LIN {X 0,Y 180.049,Z 440.205,A -85,B 0,C 180,E1 -25229.548,E2 -25229.548} C_VEL
LIN {X 0,Y 183.844,Z 448.858,A -85,B 0,C 180,E1 -25232.195,E2 -25232.195} C_VEL
LIN {X 0,Y 187.488,Z 458.143,A -85,B 0,C 180,E1 -25234.538,E2 -25234.538} C_VEL
LIN {X 0,Y 185.037,Z 489.842,A -85,B 0,C 180,E1 -25235.548,E2 -25235.548} C_VEL
LIN {X 0,Y 183.269,Z 507.581,A -85,B 0,C 180,E1 -25236.115,E2 -25236.115} C_VEL
LIN {X 0,Y 180.751,Z 522.405,A -85,B 0,C 180,E1 -25236.923,E2 -25236.923} C_VEL
LIN {X 0,Y 177.581,Z 535.216,A -85,B 0,C 180,E1 -25237.909,E2 -25237.909} C_VEL
LIN {X 0,Y 173.62,Z 547.959,A -85,B 0,C 180,E1 -25239.277,E2 -25239.277} C_VEL
LIN {X 0,Y 168.831,Z 560.376,A -85,B 0,C 180,E1 -25241.025,E2 -25241.025} C_VEL
LIN {X 0,Y 163.725,Z 571.725,A -85,B 0,C 180,E1 -25243.142,E2 -25243.142} C_VEL
LIN {X 0,Y 158.381,Z 582.164,A -85,B 0,C 180,E1 -25245.668,E2 -25245.668} C_VEL
LIN {X 0,Y 152.274,Z 592.549,A -85,B 0,C 180,E1 -25248.882,E2 -25248.882} C_VEL
LIN {X 0,Y 147.8,Z 599.416,A -85,B 0,C 180,E1 -25251.603,E2 -25251.603} C_VEL
LIN {X 0,Y 144.873,Z 602.943,A -85,B 0,C 180,E1 -25253.069,E2 -25253.069} C_VEL
LIN {X 0,Y 138.69,Z 608.311,A -85,B 0,C 180,E1 -25255.327,E2 -25255.327} C_VEL
LIN {X 0,Y 132.604,Z 613.141,A -85,B 0,C 180,E1 -25257.925,E2 -25257.925} C_VEL
LIN {X 0,Y 129.916,Z 615.782,A -85,B 0,C 180,E1 -25259.908,E2 -25259.908} C_VEL
LIN {X 0,Y 125.767,Z 621.093,A -85,B 0,C 180,E1 -25265.227,E2 -25265.227} C_VEL
LIN {X 0,Y 122.895,Z 624.585,A -85,B 0,C 180,E1 -25269.938,E2 -25269.938} C_VEL
LIN {X 0,Y 120.481,Z 627.978,A -85,B 0,C 180,E1 -25276.512,E2 -25276.512} C_VEL
LIN {X 0,Y 119.324,Z 629.978,A -85,B 0,C 180,E1 -25283.24,E2 -25283.24} C_VEL
LIN {X 0,Y 119.226,Z 630.634,A -85,B 0,C 180,E1 -25290.005,E2 -25290.005} C_VEL
LIN {X 0,Y 119.329,Z 629.948,A -85,B 0,C 180,E1 -25296.77,E2 -25296.77} C_VEL
LIN {X 0,Y 120.487,Z 627.918,A -85,B 0,C 180,E1 -25303.498,E2 -25303.498} C_VEL
LIN {X 0,Y 122.902,Z 624.501,A -85,B 0,C 180,E1 -25310.071,E2 -25310.071} C_VEL
LIN {X 0,Y 126.846,Z 619.596,A -85,B 0,C 180,E1 -25316.316,E2 -25316.316} C_VEL
LIN {X 0,Y 130.573,Z 614.948,A -85,B 0,C 180,E1 -25320.672,E2 -25320.672} C_VEL
LIN {X 0,Y 136.58,Z 608.007,A -85,B 0,C 180,E1 -25325.377,E2 -25325.377} C_VEL
LIN {X 0,Y 137.797,Z 606.89,A -85,B 0,C 180,E1 -25326.142,E2 -25326.142} C_VEL
LIN {X 0,Y 143.3,Z 607.92,A -85,B 0,C 180,E1 -25329.616,E2 -25329.616} C_VEL
LIN {X 0,Y 152.17,Z 608.59,A -85,B 0,C 180,E1 -25333.855,E2 -25333.855} C_VEL
LIN {X 0,Y 160.46,Z 608.435,A -85,B 0,C 180,E1 -25336.914,E2 -25336.914} C_VEL
LIN {X 0,Y 161.016,Z 608.309,A -85,B 0,C 180,E1 -25337.607,E2 -25337.607} C_VEL
LIN {X 0,Y 153.834,Z 607.574,A -85,B 0,C 180,E1 -25340.238,E2 -25340.238} C_VEL
LIN {X 0,Y 144.8,Z 605.575,A -85,B 0,C 180,E1 -25344.378,E2 -25344.378} C_VEL
LIN {X 0,Y 137.047,Z 602.404,A -85,B 0,C 180,E1 -25349.149,E2 -25349.149} C_VEL
LIN {X 0,Y 130.784,Z 598.022,A -85,B 0,C 180,E1 -25354.539,E2 -25354.539} C_VEL
LIN {X 0,Y 126.404,Z 592.364,A -85,B 0,C 180,E1 -25360.513,E2 -25360.513} C_VEL
LIN {X 0,Y 123.571,Z 585.19,A -85,B 0,C 180,E1 -25366.85,E2 -25366.85} C_VEL
LIN {X 0,Y 122.591,Z 577.538,A -85,B 0,C 180,E1 -25372.589,E2 -25372.589} C_VEL
LIN {X 0,Y 122.404,Z 569.444,A -85,B 0,C 180,E1 -25377.532,E2 -25377.532} C_VEL
LIN {X 0,Y 122.41,Z 566.355,A -85,B 0,C 180,E1 -25379.178,E2 -25379.178} C_VEL
LIN {X 0,Y 122.007,Z 566.876,A -85,B 0,C 180,E1 -25380,E2 -25380} C_VEL
LIN {X 0,Y 122.855,Z 565.896,A -85,B 0,C 180,E1 -25383.28,E2 -25383.28} C_VEL
LIN {X 0,Y 125.234,Z 563.196,A -85,B 0,C 180,E1 -25386.445,E2 -25386.445} C_VEL
LIN {X 0,Y 127.113,Z 561.789,A -85,B 0,C 180,E1 -25389.548,E2 -25389.548} C_VEL
LIN {X 0,Y 129.192,Z 559.973,A -85,B 0,C 180,E1 -25391.689,E2 -25391.689} C_VEL
LIN {X 0,Y 130.196,Z 558.96,A -85,B 0,C 180,E1 -25392.47,E2 -25392.47} C_VEL
LIN {X 0,Y 132.848,Z 557.281,A -85,B 0,C 180,E1 -25395.338,E2 -25395.338} C_VEL
LIN {X 0,Y 135.243,Z 555.329,A -85,B 0,C 180,E1 -25397.062,E2 -25397.062} C_VEL
LIN {X 0,Y 138.996,Z 551.77,A -85,B 0,C 180,E1 -25399.188,E2 -25399.188} C_VEL
LIN {X 0,Y 140.747,Z 550.664,A -85,B 0,C 180,E1 -25400.459,E2 -25400.459} C_VEL
LIN {X 0,Y 143.003,Z 548.959,A -85,B 0,C 180,E1 -25401.781,E2 -25401.781} C_VEL
LIN {X 0,Y 146.369,Z 545.737,A -85,B 0,C 180,E1 -25403.337,E2 -25403.337} C_VEL
LIN {X 0,Y 150.578,Z 541,A -85,B 0,C 180,E1 -25404.839,E2 -25404.839} C_VEL
LIN {X 0,Y 153.784,Z 538.288,A -85,B 0,C 180,E1 -25406.333,E2 -25406.333} C_VEL
LIN {X 0,Y 157.922,Z 533.92,A -85,B 0,C 180,E1 -25407.86,E2 -25407.86} C_VEL
LIN {X 0,Y 162.379,Z 527.957,A -85,B 0,C 180,E1 -25409.138,E2 -25409.138} C_VEL
LIN {X 0,Y 166.621,Z 520.75,A -85,B 0,C 180,E1 -25410.116,E2 -25410.116} C_VEL
LIN {X 0,Y 170.524,Z 512.516,A -85,B 0,C 180,E1 -25410.918,E2 -25410.918} C_VEL
LIN {X 0,Y 174.019,Z 506.932,A -85,B 0,C 180,E1 -25412.061,E2 -25412.061} C_VEL
LIN {X 0,Y 177.758,Z 499.232,A -85,B 0,C 180,E1 -25413.185,E2 -25413.185} C_VEL
LIN {X 0,Y 180.529,Z 491.731,A -85,B 0,C 180,E1 -25413.957,E2 -25413.957} C_VEL
LIN {X 0,Y 178.798,Z 507.903,A -85,B 0,C 180,E1 -25414.545,E2 -25414.545} C_VEL
LIN {X 0,Y 176.263,Z 521.664,A -85,B 0,C 180,E1 -25415.327,E2 -25415.327} C_VEL
LIN {X 0,Y 172.626,Z 535.679,A -85,B 0,C 180,E1 -25416.475,E2 -25416.475} C_VEL
LIN {X 0,Y 168.293,Z 548.682,A -85,B 0,C 180,E1 -25417.975,E2 -25417.975} C_VEL
LIN {X 0,Y 162.837,Z 561.826,A -85,B 0,C 180,E1 -25419.993,E2 -25419.993} C_VEL
LIN {X 0,Y 157.027,Z 573.992,A -85,B 0,C 180,E1 -25422.561,E2 -25422.561} C_VEL
LIN {X 0,Y 150.61,Z 585.153,A -85,B 0,C 180,E1 -25425.572,E2 -25425.572} C_VEL
LIN {X 0,Y 144.514,Z 594.607,A -85,B 0,C 180,E1 -25428.959,E2 -25428.959} C_VEL
LIN {X 0,Y 138.061,Z 603.617,A -85,B 0,C 180,E1 -25433.259,E2 -25433.259} C_VEL
LIN {X 0,Y 132.51,Z 610.879,A -85,B 0,C 180,E1 -25437.964,E2 -25437.964} C_VEL
LIN {X 0,Y 128.544,Z 615.963,A -85,B 0,C 180,E1 -25442.302,E2 -25442.302} C_VEL
LIN {X 0,Y 124.172,Z 621.222,A -85,B 0,C 180,E1 -25448.409,E2 -25448.409} C_VEL
LIN {X 0,Y 121.865,Z 624.157,A -85,B 0,C 180,E1 -25453.236,E2 -25453.236} C_VEL
LIN {X 0,Y 120.007,Z 626.851,A -85,B 0,C 180,E1 -25459.876,E2 -25459.876} C_VEL
LIN {X 0,Y 119.23,Z 628.198,A -85,B 0,C 180,E1 -25466.616,E2 -25466.616} C_VEL
LIN {X 0,Y 119.279,Z 628.373,A -85,B 0,C 180,E1 -25469.995,E2 -25469.995} C_VEL
LIN {X 0,Y 119.47,Z 627.741,A -85,B 0,C 180,E1 -25476.751,E2 -25476.751} C_VEL
LIN {X 0,Y 120.745,Z 625.774,A -85,B 0,C 180,E1 -25483.458,E2 -25483.458} C_VEL
LIN {X 0,Y 123.256,Z 622.422,A -85,B 0,C 180,E1 -25490,E2 -25490} C_VEL
LIN {X 0,Y 127.298,Z 617.581,A -85,B 0,C 180,E1 -25496.205,E2 -25496.205} C_VEL
LIN {X 0,Y 132.382,Z 611.11,A -85,B 0,C 180,E1 -25502.06,E2 -25502.06} C_VEL
LIN {X 0,Y 137.99,Z 603.902,A -85,B 0,C 180,E1 -25506.752,E2 -25506.752} C_VEL
LIN {X 0,Y 144.451,Z 594.978,A -85,B 0,C 180,E1 -25511.051,E2 -25511.051} C_VEL
LIN {X 0,Y 150.532,Z 585.604,A -85,B 0,C 180,E1 -25514.446,E2 -25514.446} C_VEL
LIN {X 0,Y 156.638,Z 575.089,A -85,B 0,C 180,E1 -25517.334,E2 -25517.334} C_VEL
LIN {X 0,Y 162.167,Z 563.764,A -85,B 0,C 180,E1 -25519.797,E2 -25519.797} C_VEL
LIN {X 0,Y 167.544,Z 551.06,A -85,B 0,C 180,E1 -25521.854,E2 -25521.854} C_VEL
LIN {X 0,Y 171.895,Z 538.676,A -85,B 0,C 180,E1 -25523.351,E2 -25523.351} C_VEL
LIN {X 0,Y 175.689,Z 524.933,A -85,B 0,C 180,E1 -25524.586,E2 -25524.586} C_VEL
LIN {X 0,Y 178.62,Z 510.582,A -85,B 0,C 180,E1 -25525.461,E2 -25525.461} C_VEL
LIN {X 0,Y 180.363,Z 496.588,A -85,B 0,C 180,E1 -25526.02,E2 -25526.02} C_VEL
LIN {X 0,Y 183.483,Z 458.98,A -85,B 0,C 180,E1 -25527.172,E2 -25527.172} C_VEL
LIN {X 0,Y 180.767,Z 452.209,A -85,B 0,C 180,E1 -25529.043,E2 -25529.043} C_VEL
LIN {X 0,Y 176.017,Z 443.177,A -85,B 0,C 180,E1 -25532.505,E2 -25532.505} C_VEL
LIN {X 0,Y 171.849,Z 436.037,A -85,B 0,C 180,E1 -25536.024,E2 -25536.024} C_VEL
LIN {X 0,Y 169.537,Z 432.413,A -85,B 0,C 180,E1 -25538.254,E2 -25538.254} C_VEL
LIN {X 0,Y 167.475,Z 429.194,A -85,B 0,C 180,E1 -25540.503,E2 -25540.503} C_VEL
LIN {X 0,Y 164.834,Z 425.188,A -85,B 0,C 180,E1 -25543.903,E2 -25543.903} C_VEL
LIN {X 0,Y 162.459,Z 421.538,A -85,B 0,C 180,E1 -25547.865,E2 -25547.865} C_VEL
LIN {X 0,Y 162.027,Z 420.886,A -85,B 0,C 180,E1 -25548.744,E2 -25548.744} C_VEL
LIN {X 0,Y 159.556,Z 415.986,A -85,B 0,C 180,E1 -25559.053,E2 -25559.053} C_VEL
LIN {X 0,Y 159.574,Z 415.731,A -85,B 0,C 180,E1 -25560.473,E2 -25560.473} C_VEL
LIN {X 0,Y 161.091,Z 419.996,A -85,B 0,C 180,E1 -25569.099,E2 -25569.099} C_VEL
LIN {X 0,Y 162.302,Z 421.185,A -85,B 0,C 180,E1 -25571.711,E2 -25571.711} C_VEL
LIN {X 0,Y 164.688,Z 425.102,A -85,B 0,C 180,E1 -25575.818,E2 -25575.818} C_VEL
LIN {X 0,Y 165.628,Z 426.451,A -85,B 0,C 180,E1 -25577.12,E2 -25577.12} C_VEL
LIN {X 0,Y 168.603,Z 430.922,A -85,B 0,C 180,E1 -25580.671,E2 -25580.671} C_VEL
LIN {X 0,Y 171.316,Z 435.2,A -85,B 0,C 180,E1 -25583.396,E2 -25583.396} C_VEL
LIN {X 0,Y 175.037,Z 441.482,A -85,B 0,C 180,E1 -25586.632,E2 -25586.632} C_VEL
LIN {X 0,Y 177.631,Z 446.437,A -85,B 0,C 180,E1 -25588.663,E2 -25588.663} C_VEL
LIN {X 0,Y 181.397,Z 455.639,A -85,B 0,C 180,E1 -25591.455,E2 -25591.455} C_VEL
LIN {X 0,Y 183.369,Z 460.941,A -85,B 0,C 180,E1 -25592.823,E2 -25592.823} C_VEL
LIN {X 0,Y 180.246,Z 498.172,A -85,B 0,C 180,E1 -25593.947,E2 -25593.947} C_VEL
LIN {X 0,Y 178.541,Z 512.168,A -85,B 0,C 180,E1 -25594.502,E2 -25594.502} C_VEL
LIN {X 0,Y 175.562,Z 526.623,A -85,B 0,C 180,E1 -25595.356,E2 -25595.356} C_VEL
LIN {X 0,Y 171.71,Z 540.435,A -85,B 0,C 180,E1 -25596.566,E2 -25596.566} C_VEL
LIN {X 0,Y 167.323,Z 552.871,A -85,B 0,C 180,E1 -25598.05,E2 -25598.05} C_VEL
LIN {X 0,Y 161.839,Z 565.623,A -85,B 0,C 180,E1 -25600.066,E2 -25600.066} C_VEL
LIN {X 0,Y 155.719,Z 577.908,A -85,B 0,C 180,E1 -25602.707,E2 -25602.707} C_VEL
LIN {X 0,Y 150.125,Z 587.55,A -85,B 0,C 180,E1 -25605.401,E2 -25605.401} C_VEL
LIN {X 0,Y 143.95,Z 596.966,A -85,B 0,C 180,E1 -25608.775,E2 -25608.775} C_VEL
LIN {X 0,Y 137.513,Z 605.936,A -85,B 0,C 180,E1 -25613.099,E2 -25613.099} C_VEL
LIN {X 0,Y 131.941,Z 613.186,A -85,B 0,C 180,E1 -25617.82,E2 -25617.82} C_VEL
LIN {X 0,Y 129.916,Z 615.782,A -85,B 0,C 180,E1 -25619.908,E2 -25619.908} C_VEL
LIN {X 0,Y 127.335,Z 618.257,A -85,B 0,C 180,E1 -25622.021,E2 -25622.021} C_VEL
LIN {X 0,Y 121.78,Z 621.8,A -85,B 0,C 180,E1 -25625.445,E2 -25625.445} C_VEL
LIN {X 0,Y 117.51,Z 624.222,A -85,B 0,C 180,E1 -25628.449,E2 -25628.449} C_VEL
LIN {X 0,Y 115.226,Z 625.795,A -85,B 0,C 180,E1 -25631.02,E2 -25631.02} C_VEL
LIN {X 0,Y 114.762,Z 626.273,A -85,B 0,C 180,E1 -25631.94,E2 -25631.94} C_VEL
LIN {X 0,Y 112.741,Z 629.081,A -85,B 0,C 180,E1 -25639.227,E2 -25639.227} C_VEL
LIN {X 0,Y 112.057,Z 630.405,A -85,B 0,C 180,E1 -25646.41,E2 -25646.41} C_VEL
LIN {X 0,Y 112.133,Z 630.567,A -85,B 0,C 180,E1 -25650.005,E2 -25650.005} C_VEL
LIN {X 0,Y 112.265,Z 629.88,A -85,B 0,C 180,E1 -25657.198,E2 -25657.198} C_VEL
LIN {X 0,Y 113.559,Z 627.85,A -85,B 0,C 180,E1 -25664.338,E2 -25664.338} C_VEL
LIN {X 0,Y 116.239,Z 624.433,A -85,B 0,C 180,E1 -25671.276,E2 -25671.276} C_VEL
LIN {X 0,Y 120.497,Z 619.528,A -85,B 0,C 180,E1 -25677.819,E2 -25677.819} C_VEL
LIN {X 0,Y 124.433,Z 614.974,A -85,B 0,C 180,E1 -25682.264,E2 -25682.264} C_VEL
LIN {X 0,Y 130.865,Z 607.938,A -85,B 0,C 180,E1 -25687.175,E2 -25687.175} C_VEL
LIN {X 0,Y 133.204,Z 605.542,A -85,B 0,C 180,E1 -25688.559,E2 -25688.559} C_VEL
LIN {X 0,Y 142.461,Z 607.298,A -85,B 0,C 180,E1 -25693.687,E2 -25693.687} C_VEL
LIN {X 0,Y 150.258,Z 607.914,A -85,B 0,C 180,E1 -25696.936,E2 -25696.936} C_VEL
LIN {X 0,Y 149.937,Z 607.702,A -85,B 0,C 180,E1 -25697.907,E2 -25697.907} C_VEL
LIN {X 0,Y 143.61,Z 606.297,A -85,B 0,C 180,E1 -25700.491,E2 -25700.491} C_VEL
LIN {X 0,Y 134.951,Z 603.234,A -85,B 0,C 180,E1 -25705.05,E2 -25705.05} C_VEL
LIN {X 0,Y 127.553,Z 598.977,A -85,B 0,C 180,E1 -25710.272,E2 -25710.272} C_VEL
LIN {X 0,Y 122.099,Z 593.567,A -85,B 0,C 180,E1 -25716.239,E2 -25716.239} C_VEL
LIN {X 0,Y 118.281,Z 586.7,A -85,B 0,C 180,E1 -25722.717,E2 -25722.717} C_VEL
LIN {X 0,Y 116.349,Z 578.247,A -85,B 0,C 180,E1 -25729.56,E2 -25729.56} C_VEL
LIN {X 0,Y 116.116,Z 576.393,A -85,B 0,C 180,E1 -25731.078,E2 -25731.078} C_VEL
LIN {X 0,Y 115.488,Z 576.451,A -85,B 0,C 180,E1 -25733.009,E2 -25733.009} C_VEL
LIN {X 0,Y 115.948,Z 575.011,A -85,B 0,C 180,E1 -25736.525,E2 -25736.525} C_VEL
LIN {X 0,Y 117.729,Z 572.53,A -85,B 0,C 180,E1 -25740,E2 -25740} C_VEL
LIN {X 0,Y 118.582,Z 571.656,A -85,B 0,C 180,E1 -25743.398,E2 -25743.398} C_VEL
LIN {X 0,Y 120.771,Z 569.484,A -85,B 0,C 180,E1 -25746.684,E2 -25746.684} C_VEL
LIN {X 0,Y 125.1,Z 566.252,A -85,B 0,C 180,E1 -25752.216,E2 -25752.216} C_VEL
LIN {X 0,Y 127.57,Z 564.276,A -85,B 0,C 180,E1 -25754.354,E2 -25754.354} C_VEL
LIN {X 0,Y 130.616,Z 562.473,A -85,B 0,C 180,E1 -25757.214,E2 -25757.214} C_VEL
LIN {X 0,Y 134.135,Z 559.786,A -85,B 0,C 180,E1 -25759.409,E2 -25759.409} C_VEL
LIN {X 0,Y 137.21,Z 557.185,A -85,B 0,C 180,E1 -25761.011,E2 -25761.011} C_VEL
LIN {X 0,Y 141.359,Z 554.491,A -85,B 0,C 180,E1 -25763.437,E2 -25763.437} C_VEL
LIN {X 0,Y 145.125,Z 551.29,A -85,B 0,C 180,E1 -25765.071,E2 -25765.071} C_VEL
LIN {X 0,Y 150.682,Z 545.785,A -85,B 0,C 180,E1 -25766.95,E2 -25766.95} C_VEL
LIN {X 0,Y 154.627,Z 542.586,A -85,B 0,C 180,E1 -25768.506,E2 -25768.506} C_VEL
LIN {X 0,Y 159.316,Z 537.762,A -85,B 0,C 180,E1 -25769.975,E2 -25769.975} C_VEL
LIN {X 0,Y 164.357,Z 531.357,A -85,B 0,C 180,E1 -25771.211,E2 -25771.211} C_VEL
LIN {X 0,Y 168.738,Z 524.439,A -85,B 0,C 180,E1 -25772.075,E2 -25772.075} C_VEL
LIN {X 0,Y 172.959,Z 516.311,A -85,B 0,C 180,E1 -25772.812,E2 -25772.812} C_VEL
LIN {X 0,Y 173.507,Z 515.542,A -85,B 0,C 180,E1 -25772.98,E2 -25772.98} C_VEL
LIN {X 0,Y 170.155,Z 530.121,A -85,B 0,C 180,E1 -25774.034,E2 -25774.034} C_VEL
LIN {X 0,Y 165.901,Z 543.532,A -85,B 0,C 180,E1 -25775.36,E2 -25775.36} C_VEL
LIN {X 0,Y 160.865,Z 556.404,A -85,B 0,C 180,E1 -25777.12,E2 -25777.12} C_VEL
LIN {X 0,Y 155.854,Z 567.153,A -85,B 0,C 180,E1 -25779.033,E2 -25779.033} C_VEL
LIN {X 0,Y 150.17,Z 577.805,A -85,B 0,C 180,E1 -25781.508,E2 -25781.508} C_VEL
LIN {X 0,Y 144.502,Z 586.928,A -85,B 0,C 180,E1 -25784.156,E2 -25784.156} C_VEL
LIN {X 0,Y 138.201,Z 596.071,A -85,B 0,C 180,E1 -25787.633,E2 -25787.633} C_VEL
LIN {X 0,Y 131.516,Z 604.8,A -85,B 0,C 180,E1 -25792.076,E2 -25792.076} C_VEL
LIN {X 0,Y 125.759,Z 611.832,A -85,B 0,C 180,E1 -25796.959,E2 -25796.959} C_VEL
LIN {X 0,Y 121.001,Z 617.469,A -85,B 0,C 180,E1 -25802.307,E2 -25802.307} C_VEL
LIN {X 0,Y 116.609,Z 622.351,A -85,B 0,C 180,E1 -25808.795,E2 -25808.795} C_VEL
LIN {X 0,Y 113.846,Z 625.745,A -85,B 0,C 180,E1 -25815.699,E2 -25815.699} C_VEL
LIN {X 0,Y 112.437,Z 627.758,A -85,B 0,C 180,E1 -25822.813,E2 -25822.813} C_VEL
LIN {X 0,Y 112.199,Z 628.441,A -85,B 0,C 180,E1 -25829.995,E2 -25829.995} C_VEL
LIN {X 0,Y 112.432,Z 627.808,A -85,B 0,C 180,E1 -25837.176,E2 -25837.176} C_VEL
LIN {X 0,Y 113.816,Z 625.841,A -85,B 0,C 180,E1 -25844.294,E2 -25844.294} C_VEL
LIN {X 0,Y 116.577,Z 622.489,A -85,B 0,C 180,E1 -25851.2,E2 -25851.2} C_VEL
LIN {X 0,Y 120.918,Z 617.647,A -85,B 0,C 180,E1 -25857.703,E2 -25857.703} C_VEL
LIN {X 0,Y 126.402,Z 611.176,A -85,B 0,C 180,E1 -25863.774,E2 -25863.774} C_VEL
LIN {X 0,Y 132.35,Z 603.967,A -85,B 0,C 180,E1 -25868.598,E2 -25868.598} C_VEL
LIN {X 0,Y 139.154,Z 595.044,A -85,B 0,C 180,E1 -25872.98,E2 -25872.98} C_VEL
LIN {X 0,Y 145.542,Z 585.668,A -85,B 0,C 180,E1 -25876.406,E2 -25876.406} C_VEL
LIN {X 0,Y 151.724,Z 575.483,A -85,B 0,C 180,E1 -25879.231,E2 -25879.231} C_VEL
LIN {X 0,Y 157.072,Z 565.117,A -85,B 0,C 180,E1 -25881.531,E2 -25881.531} C_VEL
LIN {X 0,Y 162.622,Z 552.702,A -85,B 0,C 180,E1 -25883.594,E2 -25883.594} C_VEL
LIN {X 0,Y 167.113,Z 540.724,A -85,B 0,C 180,E1 -25885.085,E2 -25885.085} C_VEL
LIN {X 0,Y 171.038,Z 527.591,A -85,B 0,C 180,E1 -25886.305,E2 -25886.305} C_VEL
LIN {X 0,Y 174.2,Z 513.38,A -85,B 0,C 180,E1 -25887.231,E2 -25887.231} C_VEL
LIN {X 0,Y 176.218,Z 499.187,A -85,B 0,C 180,E1 -25887.848,E2 -25887.848} C_VEL
LIN {X 0,Y 179.534,Z 461.909,A -85,B 0,C 180,E1 -25888.96,E2 -25888.96} C_VEL
LIN {X 0,Y 177.486,Z 456.701,A -85,B 0,C 180,E1 -25890.496,E2 -25890.496} C_VEL
LIN {X 0,Y 173.099,Z 448.164,A -85,B 0,C 180,E1 -25893.96,E2 -25893.96} C_VEL
LIN {X 0,Y 169.507,Z 441.747,A -85,B 0,C 180,E1 -25897.254,E2 -25897.254} C_VEL
LIN {X 0,Y 166.136,Z 436.061,A -85,B 0,C 180,E1 -25900.942,E2 -25900.942} C_VEL
LIN {X 0,Y 163.407,Z 431.873,A -85,B 0,C 180,E1 -25904.617,E2 -25904.617} C_VEL
LIN {X 0,Y 161.156,Z 428.124,A -85,B 0,C 180,E1 -25908.682,E2 -25908.682} C_VEL
LIN {X 0,Y 158.709,Z 422.73,A -85,B 0,C 180,E1 -25920,E2 -25920} C_VEL
LIN {X 0,Y 161.187,Z 428.257,A -85,B 0,C 180,E1 -25931.315,E2 -25931.315} C_VEL
LIN {X 0,Y 163.993,Z 432.815,A -85,B 0,C 180,E1 -25936.17,E2 -25936.17} C_VEL
LIN {X 0,Y 166.867,Z 437.39,A -85,B 0,C 180,E1 -25939.851,E2 -25939.851} C_VEL
LIN {X 0,Y 169.724,Z 442.106,A -85,B 0,C 180,E1 -25942.871,E2 -25942.871} C_VEL
LIN {X 0,Y 173.841,Z 449.463,A -85,B 0,C 180,E1 -25946.566,E2 -25946.566} C_VEL
LIN {X 0,Y 176.926,Z 456.928,A -85,B 0,C 180,E1 -25949.111,E2 -25949.111} C_VEL
LIN {X 0,Y 179.409,Z 463.663,A -85,B 0,C 180,E1 -25951.018,E2 -25951.018} C_VEL
LIN {X 0,Y 175.521,Z 505.752,A -85,B 0,C 180,E1 -25952.287,E2 -25952.287} C_VEL
LIN {X 0,Y 173.121,Z 520.004,A -85,B 0,C 180,E1 -25953.019,E2 -25953.019} C_VEL
LIN {X 0,Y 169.572,Z 533.965,A -85,B 0,C 180,E1 -25954.02,E2 -25954.02} C_VEL
LIN {X 0,Y 165.61,Z 546.068,A -85,B 0,C 180,E1 -25955.231,E2 -25955.231} C_VEL
LIN {X 0,Y 160.495,Z 558.824,A -85,B 0,C 180,E1 -25956.957,E2 -25956.957} C_VEL
LIN {X 0,Y 154.917,Z 570.423,A -85,B 0,C 180,E1 -25959.03,E2 -25959.03} C_VEL
LIN {X 0,Y 148.511,Z 582.035,A -85,B 0,C 180,E1 -25961.819,E2 -25961.819} C_VEL
LIN {X 0,Y 141.861,Z 592.419,A -85,B 0,C 180,E1 -25965.099,E2 -25965.099} C_VEL
LIN {X 0,Y 135.669,Z 600.986,A -85,B 0,C 180,E1 -25968.67,E2 -25968.67} C_VEL
LIN {X 0,Y 129.223,Z 609.185,A -85,B 0,C 180,E1 -25973.262,E2 -25973.262} C_VEL
LIN {X 0,Y 123.341,Z 616.231,A -85,B 0,C 180,E1 -25978.726,E2 -25978.726} C_VEL
LIN {X 0,Y 119.301,Z 621.026,A -85,B 0,C 180,E1 -25983.786,E2 -25983.786} C_VEL
LIN {X 0,Y 116.233,Z 624.519,A -85,B 0,C 180,E1 -25988.734,E2 -25988.734} C_VEL
LIN {X 0,Y 114.762,Z 626.273,A -85,B 0,C 180,E1 -25991.94,E2 -25991.94} C_VEL
LIN {X 0,Y 113.119,Z 627.638,A -85,B 0,C 180,E1 -25994.71,E2 -25994.71} C_VEL
LIN {X 0,Y 109.144,Z 629.254,A -85,B 0,C 180,E1 -25999.321,E2 -25999.321} C_VEL
LIN {X 0,Y 106.219,Z 630.024,A -85,B 0,C 180,E1 -26003.261,E2 -26003.261} C_VEL
LIN {X 0,Y 105.025,Z 630.357,A -85,B 0,C 180,E1 -26006.425,E2 -26006.425} C_VEL
LIN {X 0,Y 104.933,Z 630.394,A -85,B 0,C 180,E1 -26007.507,E2 -26007.507} C_VEL
LIN {X 0,Y 105.033,Z 630.499,A -85,B 0,C 180,E1 -26010.006,E2 -26010.006} C_VEL
LIN {X 0,Y 105.223,Z 629.812,A -85,B 0,C 180,E1 -26017.682,E2 -26017.682} C_VEL
LIN {X 0,Y 106.645,Z 627.782,A -85,B 0,C 180,E1 -26025.29,E2 -26025.29} C_VEL
LIN {X 0,Y 109.636,Z 624.364,A -85,B 0,C 180,E1 -26032.626,E2 -26032.626} C_VEL
LIN {X 0,Y 114.241,Z 619.459,A -85,B 0,C 180,E1 -26039.488,E2 -26039.488} C_VEL
LIN {X 0,Y 118.647,Z 614.726,A -85,B 0,C 180,E1 -26044.248,E2 -26044.248} C_VEL
LIN {X 0,Y 125.276,Z 607.869,A -85,B 0,C 180,E1 -26049.139,E2 -26049.139} C_VEL
LIN {X 0,Y 129.047,Z 604.118,A -85,B 0,C 180,E1 -26051.201,E2 -26051.201} C_VEL
LIN {X 0,Y 140.29,Z 606.401,A -85,B 0,C 180,E1 -26056.912,E2 -26056.912} C_VEL
LIN {X 0,Y 139.822,Z 606.117,A -85,B 0,C 180,E1 -26057.956,E2 -26057.956} C_VEL
LIN {X 0,Y 129.277,Z 602.077,A -85,B 0,C 180,E1 -26063.273,E2 -26063.273} C_VEL
LIN {X 0,Y 121.621,Z 597.35,A -85,B 0,C 180,E1 -26068.663,E2 -26068.663} C_VEL
LIN {X 0,Y 115.928,Z 591.488,A -85,B 0,C 180,E1 -26074.89,E2 -26074.89} C_VEL
LIN {X 0,Y 112.573,Z 586.104,A -85,B 0,C 180,E1 -26080.19,E2 -26080.19} C_VEL
LIN {X 0,Y 111.543,Z 586.122,A -85,B 0,C 180,E1 -26081.637,E2 -26081.637} C_VEL
LIN {X 0,Y 110.392,Z 585.152,A -85,B 0,C 180,E1 -26085.247,E2 -26085.247} C_VEL
LIN {X 0,Y 110.82,Z 581.741,A -85,B 0,C 180,E1 -26092.713,E2 -26092.713} C_VEL
LIN {X 0,Y 111.167,Z 580.54,A -85,B 0,C 180,E1 -26096.376,E2 -26096.376} C_VEL
LIN {X 0,Y 112.723,Z 578.497,A -85,B 0,C 180,E1 -26100,E2 -26100} C_VEL
LIN {X 0,Y 114.037,Z 577.203,A -85,B 0,C 180,E1 -26103.534,E2 -26103.534} C_VEL
LIN {X 0,Y 121.396,Z 571.801,A -85,B 0,C 180,E1 -26113.39,E2 -26113.39} C_VEL
LIN {X 0,Y 124.884,Z 569.423,A -85,B 0,C 180,E1 -26116.343,E2 -26116.343} C_VEL
LIN {X 0,Y 128.339,Z 567.515,A -85,B 0,C 180,E1 -26119.182,E2 -26119.182} C_VEL
LIN {X 0,Y 132.92,Z 564.256,A -85,B 0,C 180,E1 -26121.723,E2 -26121.723} C_VEL
LIN {X 0,Y 135.379,Z 562.435,A -85,B 0,C 180,E1 -26122.915,E2 -26122.915} C_VEL
LIN {X 0,Y 139.985,Z 559.631,A -85,B 0,C 180,E1 -26125.343,E2 -26125.343} C_VEL
LIN {X 0,Y 144.888,Z 555.809,A -85,B 0,C 180,E1 -26127.232,E2 -26127.232} C_VEL
LIN {X 0,Y 149.876,Z 551.225,A -85,B 0,C 180,E1 -26128.728,E2 -26128.728} C_VEL
LIN {X 0,Y 154.971,Z 547.24,A -85,B 0,C 180,E1 -26130.49,E2 -26130.49} C_VEL
LIN {X 0,Y 160.632,Z 541.796,A -85,B 0,C 180,E1 -26132.019,E2 -26132.019} C_VEL
LIN {X 0,Y 162.793,Z 539.338,A -85,B 0,C 180,E1 -26132.517,E2 -26132.517} C_VEL
LIN {X 0,Y 162.9,Z 540.828,A -85,B 0,C 180,E1 -26133.007,E2 -26133.007} C_VEL
LIN {X 0,Y 157.982,Z 553.566,A -85,B 0,C 180,E1 -26134.609,E2 -26134.609} C_VEL
LIN {X 0,Y 152.217,Z 565.812,A -85,B 0,C 180,E1 -26136.651,E2 -26136.651} C_VEL
LIN {X 0,Y 145.556,Z 577.876,A -85,B 0,C 180,E1 -26139.412,E2 -26139.412} C_VEL
LIN {X 0,Y 139.647,Z 586.998,A -85,B 0,C 180,E1 -26142.065,E2 -26142.065} C_VEL
LIN {X 0,Y 133.033,Z 596.14,A -85,B 0,C 180,E1 -26145.569,E2 -26145.569} C_VEL
LIN {X 0,Y 125.967,Z 604.869,A -85,B 0,C 180,E1 -26150.082,E2 -26150.082} C_VEL
LIN {X 0,Y 119.51,Z 612.278,A -85,B 0,C 180,E1 -26155.417,E2 -26155.417} C_VEL
LIN {X 0,Y 114.719,Z 617.538,A -85,B 0,C 180,E1 -26160.647,E2 -26160.647} C_VEL
LIN {X 0,Y 109.988,Z 622.419,A -85,B 0,C 180,E1 -26167.451,E2 -26167.451} C_VEL
LIN {X 0,Y 106.953,Z 625.813,A -85,B 0,C 180,E1 -26174.755,E2 -26174.755} C_VEL
LIN {X 0,Y 105.38,Z 627.826,A -85,B 0,C 180,E1 -26182.329,E2 -26182.329} C_VEL
LIN {X 0,Y 105.106,Z 628.508,A -85,B 0,C 180,E1 -26189.994,E2 -26189.994} C_VEL
LIN {X 0,Y 105.371,Z 627.875,A -85,B 0,C 180,E1 -26197.66,E2 -26197.66} C_VEL
LIN {X 0,Y 106.925,Z 625.908,A -85,B 0,C 180,E1 -26205.237,E2 -26205.237} C_VEL
LIN {X 0,Y 109.956,Z 622.555,A -85,B 0,C 180,E1 -26212.544,E2 -26212.544} C_VEL
LIN {X 0,Y 114.633,Z 617.714,A -85,B 0,C 180,E1 -26219.365,E2 -26219.365} C_VEL
LIN {X 0,Y 120.545,Z 611.242,A -85,B 0,C 180,E1 -26225.656,E2 -26225.656} C_VEL
LIN {X 0,Y 126.859,Z 604.033,A -85,B 0,C 180,E1 -26230.607,E2 -26230.607} C_VEL
LIN {X 0,Y 134.012,Z 595.109,A -85,B 0,C 180,E1 -26235.064,E2 -26235.064} C_VEL
LIN {X 0,Y 140.733,Z 585.733,A -85,B 0,C 180,E1 -26238.503,E2 -26238.503} C_VEL
LIN {X 0,Y 147.001,Z 575.855,A -85,B 0,C 180,E1 -26241.256,E2 -26241.256} C_VEL
LIN {X 0,Y 152.742,Z 565.18,A -85,B 0,C 180,E1 -26243.623,E2 -26243.623} C_VEL
LIN {X 0,Y 158.514,Z 552.764,A -85,B 0,C 180,E1 -26245.659,E2 -26245.659} C_VEL
LIN {X 0,Y 163.15,Z 540.785,A -85,B 0,C 180,E1 -26247.132,E2 -26247.132} C_VEL
LIN {X 0,Y 167.199,Z 527.649,A -85,B 0,C 180,E1 -26248.333,E2 -26248.333} C_VEL
LIN {X 0,Y 170.47,Z 513.436,A -85,B 0,C 180,E1 -26249.233,E2 -26249.233} C_VEL
LIN {X 0,Y 172.534,Z 499.358,A -85,B 0,C 180,E1 -26249.838,E2 -26249.838} C_VEL
LIN {X 0,Y 175.743,Z 464.731,A -85,B 0,C 180,E1 -26250.851,E2 -26250.851} C_VEL
LIN {X 0,Y 173.354,Z 459.279,A -85,B 0,C 180,E1 -26252.783,E2 -26252.783} C_VEL
LIN {X 0,Y 169.699,Z 451.946,A -85,B 0,C 180,E1 -26256.034,E2 -26256.034} C_VEL
LIN {X 0,Y 166.409,Z 445.917,A -85,B 0,C 180,E1 -26259.447,E2 -26259.447} C_VEL
LIN {X 0,Y 164.118,Z 442.099,A -85,B 0,C 180,E1 -26262.235,E2 -26262.235} C_VEL
LIN {X 0,Y 161.974,Z 438.524,A -85,B 0,C 180,E1 -26265.392,E2 -26265.392} C_VEL
LIN {X 0,Y 159.72,Z 434.628,A -85,B 0,C 180,E1 -26269.862,E2 -26269.862} C_VEL
LIN {X 0,Y 157.829,Z 429.894,A -85,B 0,C 180,E1 -26280,E2 -26280} C_VEL
LIN {X 0,Y 160.006,Z 435.091,A -85,B 0,C 180,E1 -26290.719,E2 -26290.719} C_VEL
LIN {X 0,Y 162.694,Z 439.742,A -85,B 0,C 180,E1 -26295.661,E2 -26295.661} C_VEL
LIN {X 0,Y 165.227,Z 443.956,A -85,B 0,C 180,E1 -26299.086,E2 -26299.086} C_VEL
LIN {X 0,Y 167.938,Z 448.676,A -85,B 0,C 180,E1 -26302.125,E2 -26302.125} C_VEL
LIN {X 0,Y 171.661,Z 455.806,A -85,B 0,C 180,E1 -26305.68,E2 -26305.68} C_VEL
LIN {X 0,Y 174.461,Z 463.246,A -85,B 0,C 180,E1 -26308.169,E2 -26308.169} C_VEL
LIN {X 0,Y 175.577,Z 466.452,A -85,B 0,C 180,E1 -26309.106,E2 -26309.106} C_VEL
LIN {X 0,Y 171.984,Z 504.535,A -85,B 0,C 180,E1 -26310.235,E2 -26310.235} C_VEL
LIN {X 0,Y 169.71,Z 518.412,A -85,B 0,C 180,E1 -26310.915,E2 -26310.915} C_VEL
LIN {X 0,Y 166.035,Z 532.775,A -85,B 0,C 180,E1 -26311.882,E2 -26311.882} C_VEL
LIN {X 0,Y 161.626,Z 546.006,A -85,B 0,C 180,E1 -26313.178,E2 -26313.178} C_VEL
LIN {X 0,Y 156.332,Z 558.761,A -85,B 0,C 180,E1 -26314.879,E2 -26314.879} C_VEL
LIN {X 0,Y 150.538,Z 570.359,A -85,B 0,C 180,E1 -26316.926,E2 -26316.926} C_VEL
LIN {X 0,Y 143.862,Z 581.97,A -85,B 0,C 180,E1 -26319.705,E2 -26319.705} C_VEL
LIN {X 0,Y 136.903,Z 592.354,A -85,B 0,C 180,E1 -26322.992,E2 -26322.992} C_VEL
LIN {X 0,Y 130.393,Z 600.921,A -85,B 0,C 180,E1 -26326.598,E2 -26326.598} C_VEL
LIN {X 0,Y 123.568,Z 609.119,A -85,B 0,C 180,E1 -26331.278,E2 -26331.278} C_VEL
LIN {X 0,Y 118.488,Z 614.866,A -85,B 0,C 180,E1 -26335.71,E2 -26335.71} C_VEL
LIN {X 0,Y 114.213,Z 619.571,A -85,B 0,C 180,E1 -26340.516,E2 -26340.516} C_VEL
LIN {X 0,Y 109.63,Z 624.452,A -85,B 0,C 180,E1 -26347.385,E2 -26347.385} C_VEL
LIN {X 0,Y 106.639,Z 627.843,A -85,B 0,C 180,E1 -26354.721,E2 -26354.721} C_VEL
LIN {X 0,Y 105.218,Z 629.844,A -85,B 0,C 180,E1 -26362.329,E2 -26362.329} C_VEL
LIN {X 0,Y 104.933,Z 630.394,A -85,B 0,C 180,E1 -26367.507,E2 -26367.507} C_VEL
LIN {X 0,Y 104.271,Z 630.467,A -85,B 0,C 180,E1 -26370.712,E2 -26370.712} C_VEL
LIN {X 0,Y 102.753,Z 630.306,A -85,B 0,C 180,E1 -26373.892,E2 -26373.892} C_VEL
LIN {X 0,Y 99.589,Z 629.296,A -85,B 0,C 180,E1 -26380.451,E2 -26380.451} C_VEL
LIN {X 0,Y 99.182,Z 628.468,A -85,B 0,C 180,E1 -26383.869,E2 -26383.869} C_VEL
LIN {X 0,Y 99.38,Z 628.118,A -85,B 0,C 180,E1 -26385.003,E2 -26385.003} C_VEL
LIN {X 0,Y 101.17,Z 626.183,A -85,B 0,C 180,E1 -26390.331,E2 -26390.331} C_VEL
LIN {X 0,Y 105.391,Z 622.038,A -85,B 0,C 180,E1 -26397.833,E2 -26397.833} C_VEL
LIN {X 0,Y 111.094,Z 616.332,A -85,B 0,C 180,E1 -26404.711,E2 -26404.711} C_VEL
LIN {X 0,Y 117.692,Z 609.903,A -85,B 0,C 180,E1 -26409.942,E2 -26409.942} C_VEL
LIN {X 0,Y 125.037,Z 602.7,A -85,B 0,C 180,E1 -26413.939,E2 -26413.939} C_VEL
LIN {X 0,Y 130.645,Z 603.964,A -85,B 0,C 180,E1 -26416.859,E2 -26416.859} C_VEL
LIN {X 0,Y 130.03,Z 603.582,A -85,B 0,C 180,E1 -26418.01,E2 -26418.01} C_VEL
LIN {X 0,Y 121.641,Z 599.508,A -85,B 0,C 180,E1 -26422.652,E2 -26422.652} C_VEL
LIN {X 0,Y 114.372,Z 594.26,A -85,B 0,C 180,E1 -26428.254,E2 -26428.254} C_VEL
LIN {X 0,Y 112.327,Z 594.236,A -85,B 0,C 180,E1 -26429.965,E2 -26429.965} C_VEL
LIN {X 0,Y 109.076,Z 593.167,A -85,B 0,C 180,E1 -26434.44,E2 -26434.44} C_VEL
LIN {X 0,Y 106.665,Z 591.007,A -85,B 0,C 180,E1 -26440.765,E2 -26440.765} C_VEL
LIN {X 0,Y 105.369,Z 590.161,A -85,B 0,C 180,E1 -26444.527,E2 -26444.527} C_VEL
LIN {X 0,Y 105.928,Z 586.317,A -85,B 0,C 180,E1 -26454.44,E2 -26454.44} C_VEL
LIN {X 0,Y 106.146,Z 585.794,A -85,B 0,C 180,E1 -26456.204,E2 -26456.204} C_VEL
LIN {X 0,Y 109.142,Z 582.613,A -85,B 0,C 180,E1 -26463.692,E2 -26463.692} C_VEL
LIN {X 0,Y 115.008,Z 578.553,A -85,B 0,C 180,E1 -26472.09,E2 -26472.09} C_VEL
LIN {X 0,Y 126.032,Z 572.402,A -85,B 0,C 180,E1 -26481.252,E2 -26481.252} C_VEL
LIN {X 0,Y 133.52,Z 567.519,A -85,B 0,C 180,E1 -26484.904,E2 -26484.904} C_VEL
LIN {X 0,Y 138.326,Z 564.796,A -85,B 0,C 180,E1 -26487.211,E2 -26487.211} C_VEL
LIN {X 0,Y 144.009,Z 560.789,A -85,B 0,C 180,E1 -26489.211,E2 -26489.211} C_VEL
LIN {X 0,Y 150.316,Z 555.563,A -85,B 0,C 180,E1 -26490.951,E2 -26490.951} C_VEL
LIN {X 0,Y 153.94,Z 552.944,A -85,B 0,C 180,E1 -26492.092,E2 -26492.092} C_VEL
LIN {X 0,Y 153.507,Z 554.88,A -85,B 0,C 180,E1 -26492.616,E2 -26492.616} C_VEL
LIN {X 0,Y 147.436,Z 567.059,A -85,B 0,C 180,E1 -26494.681,E2 -26494.681} C_VEL
LIN {X 0,Y 141.156,Z 577.946,A -85,B 0,C 180,E1 -26497.185,E2 -26497.185} C_VEL
LIN {X 0,Y 133.776,Z 588.693,A -85,B 0,C 180,E1 -26500.374,E2 -26500.374} C_VEL
LIN {X 0,Y 126.93,Z 597.561,A -85,B 0,C 180,E1 -26503.956,E2 -26503.956} C_VEL
LIN {X 0,Y 119.589,Z 606.052,A -85,B 0,C 180,E1 -26508.607,E2 -26508.607} C_VEL
LIN {X 0,Y 113.294,Z 612.78,A -85,B 0,C 180,E1 -26513.75,E2 -26513.75} C_VEL
LIN {X 0,Y 108.547,Z 617.607,A -85,B 0,C 180,E1 -26518.798,E2 -26518.798} C_VEL
LIN {X 0,Y 103.437,Z 622.487,A -85,B 0,C 180,E1 -26525.936,E2 -26525.936} C_VEL
LIN {X 0,Y 100.101,Z 625.881,A -85,B 0,C 180,E1 -26533.684,E2 -26533.684} C_VEL
LIN {X 0,Y 98.338,Z 627.893,A -85,B 0,C 180,E1 -26541.776,E2 -26541.776} C_VEL
LIN {X 0,Y 98.006,Z 628.575,A -85,B 0,C 180,E1 -26549.994,E2 -26549.994} C_VEL
LIN {X 0,Y 98.329,Z 627.942,A -85,B 0,C 180,E1 -26558.212,E2 -26558.212} C_VEL
LIN {X 0,Y 100.076,Z 625.975,A -85,B 0,C 180,E1 -26566.308,E2 -26566.308} C_VEL
LIN {X 0,Y 103.407,Z 622.622,A -85,B 0,C 180,E1 -26574.059,E2 -26574.059} C_VEL
LIN {X 0,Y 108.46,Z 617.78,A -85,B 0,C 180,E1 -26581.217,E2 -26581.217} C_VEL
LIN {X 0,Y 114.813,Z 611.309,A -85,B 0,C 180,E1 -26587.736,E2 -26587.736} C_VEL
LIN {X 0,Y 121.546,Z 604.099,A -85,B 0,C 180,E1 -26592.79,E2 -26592.79} C_VEL
LIN {X 0,Y 129.07,Z 595.174,A -85,B 0,C 180,E1 -26597.307,E2 -26597.307} C_VEL
LIN {X 0,Y 136.126,Z 585.797,A -85,B 0,C 180,E1 -26600.746,E2 -26600.746} C_VEL
LIN {X 0,Y 143.347,Z 574.691,A -85,B 0,C 180,E1 -26603.793,E2 -26603.793} C_VEL
LIN {X 0,Y 149.309,Z 563.954,A -85,B 0,C 180,E1 -26606.051,E2 -26606.051} C_VEL
LIN {X 0,Y 154.616,Z 552.827,A -85,B 0,C 180,E1 -26607.834,E2 -26607.834} C_VEL
LIN {X 0,Y 159.41,Z 540.846,A -85,B 0,C 180,E1 -26609.275,E2 -26609.275} C_VEL
LIN {X 0,Y 163.551,Z 527.829,A -85,B 0,C 180,E1 -26610.44,E2 -26610.44} C_VEL
LIN {X 0,Y 167.022,Z 513.17,A -85,B 0,C 180,E1 -26611.337,E2 -26611.337} C_VEL
LIN {X 0,Y 169.043,Z 499.804,A -85,B 0,C 180,E1 -26611.899,E2 -26611.899} C_VEL
LIN {X 0,Y 172.116,Z 467.779,A -85,B 0,C 180,E1 -26612.825,E2 -26612.825} C_VEL
LIN {X 0,Y 168.398,Z 459.707,A -85,B 0,C 180,E1 -26616.232,E2 -26616.232} C_VEL
LIN {X 0,Y 164.99,Z 452.952,A -85,B 0,C 180,E1 -26619.913,E2 -26619.913} C_VEL
LIN {X 0,Y 162.426,Z 448.43,A -85,B 0,C 180,E1 -26623.228,E2 -26623.228} C_VEL
LIN {X 0,Y 160.546,Z 445.111,A -85,B 0,C 180,E1 -26626.229,E2 -26626.229} C_VEL
LIN {X 0,Y 158.657,Z 441.539,A -85,B 0,C 180,E1 -26630.277,E2 -26630.277} C_VEL
LIN {X 0,Y 156.946,Z 437.086,A -85,B 0,C 180,E1 -26640,E2 -26640} C_VEL
LIN {X 0,Y 158.871,Z 441.999,A -85,B 0,C 180,E1 -26650.192,E2 -26650.192} C_VEL
LIN {X 0,Y 161.178,Z 446.207,A -85,B 0,C 180,E1 -26654.762,E2 -26654.762} C_VEL
LIN {X 0,Y 163.647,Z 450.559,A -85,B 0,C 180,E1 -26658.343,E2 -26658.343} C_VEL
LIN {X 0,Y 166.393,Z 455.686,A -85,B 0,C 180,E1 -26661.599,E2 -26661.599} C_VEL
LIN {X 0,Y 169.395,Z 461.887,A -85,B 0,C 180,E1 -26664.652,E2 -26664.652} C_VEL
LIN {X 0,Y 171.993,Z 469.449,A -85,B 0,C 180,E1 -26667.157,E2 -26667.157} C_VEL
LIN {X 0,Y 168.361,Z 505.645,A -85,B 0,C 180,E1 -26668.195,E2 -26668.195} C_VEL
LIN {X 0,Y 165.9,Z 519.533,A -85,B 0,C 180,E1 -26668.884,E2 -26668.884} C_VEL
LIN {X 0,Y 162.048,Z 533.845,A -85,B 0,C 180,E1 -26669.851,E2 -26669.851} C_VEL
LIN {X 0,Y 157.16,Z 547.712,A -85,B 0,C 180,E1 -26671.221,E2 -26671.221} C_VEL
LIN {X 0,Y 151.7,Z 560.125,A -85,B 0,C 180,E1 -26672.9,E2 -26672.9} C_VEL
LIN {X 0,Y 145.728,Z 571.47,A -85,B 0,C 180,E1 -26674.938,E2 -26674.938} C_VEL
LIN {X 0,Y 139.426,Z 581.906,A -85,B 0,C 180,E1 -26677.456,E2 -26677.456} C_VEL
LIN {X 0,Y 132.143,Z 592.289,A -85,B 0,C 180,E1 -26680.73,E2 -26680.73} C_VEL
LIN {X 0,Y 125.307,Z 600.855,A -85,B 0,C 180,E1 -26684.356,E2 -26684.356} C_VEL
LIN {X 0,Y 118.092,Z 609.053,A -85,B 0,C 180,E1 -26689.115,E2 -26689.115} C_VEL
LIN {X 0,Y 112.641,Z 614.8,A -85,B 0,C 180,E1 -26693.656,E2 -26693.656} C_VEL
LIN {X 0,Y 106.657,Z 620.893,A -85,B 0,C 180,E1 -26700.39,E2 -26700.39} C_VEL
LIN {X 0,Y 103.095,Z 624.385,A -85,B 0,C 180,E1 -26705.864,E2 -26705.864} C_VEL
LIN {X 0,Y 99.765,Z 627.776,A -85,B 0,C 180,E1 -26713.64,E2 -26713.64} C_VEL
LIN {X 0,Y 98.175,Z 629.777,A -85,B 0,C 180,E1 -26721.775,E2 -26721.775} C_VEL
LIN {X 0,Y 97.94,Z 630.432,A -85,B 0,C 180,E1 -26730.006,E2 -26730.006} C_VEL
LIN {X 0,Y 98.18,Z 629.745,A -85,B 0,C 180,E1 -26738.237,E2 -26738.237} C_VEL
LIN {X 0,Y 99.38,Z 628.118,A -85,B 0,C 180,E1 -26745.003,E2 -26745.003} C_VEL
LIN {X 0,Y 99.743,Z 627.054,A -85,B 0,C 180,E1 -26748.345,E2 -26748.345} C_VEL
LIN {X 0,Y 99.231,Z 624.905,A -85,B 0,C 180,E1 -26753.924,E2 -26753.924} C_VEL
LIN {X 0,Y 99.575,Z 622.132,A -85,B 0,C 180,E1 -26759.42,E2 -26759.42} C_VEL
LIN {X 0,Y 101.21,Z 620.092,A -85,B 0,C 180,E1 -26762.449,E2 -26762.449} C_VEL
LIN {X 0,Y 105.313,Z 616.263,A -85,B 0,C 180,E1 -26766.92,E2 -26766.92} C_VEL
LIN {X 0,Y 112.337,Z 609.834,A -85,B 0,C 180,E1 -26772.27,E2 -26772.27} C_VEL
LIN {X 0,Y 120.8,Z 601.861,A -85,B 0,C 180,E1 -26776.662,E2 -26776.662} C_VEL
LIN {X 0,Y 120.197,Z 600.56,A -85,B 0,C 180,E1 -26778.209,E2 -26778.209} C_VEL
LIN {X 0,Y 114.146,Z 600.21,A -85,B 0,C 180,E1 -26781.997,E2 -26781.997} C_VEL
LIN {X 0,Y 109.753,Z 599.017,A -85,B 0,C 180,E1 -26786.36,E2 -26786.36} C_VEL
LIN {X 0,Y 104.754,Z 598.049,A -85,B 0,C 180,E1 -26791.99,E2 -26791.99} C_VEL
LIN {X 0,Y 101.452,Z 595.779,A -85,B 0,C 180,E1 -26799.735,E2 -26799.735} C_VEL
LIN {X 0,Y 100.165,Z 594.893,A -85,B 0,C 180,E1 -26803.701,E2 -26803.701} C_VEL
LIN {X 0,Y 106.585,Z 586.061,A -85,B 0,C 180,E1 -26828.445,E2 -26828.445} C_VEL
LIN {X 0,Y 115.464,Z 581.185,A -85,B 0,C 180,E1 -26837.719,E2 -26837.719} C_VEL
LIN {X 0,Y 123.719,Z 577.128,A -85,B 0,C 180,E1 -26843.431,E2 -26843.431} C_VEL
LIN {X 0,Y 131.647,Z 572.444,A -85,B 0,C 180,E1 -26846.986,E2 -26846.986} C_VEL
LIN {X 0,Y 137.057,Z 569.574,A -85,B 0,C 180,E1 -26849.332,E2 -26849.332} C_VEL
LIN {X 0,Y 143.177,Z 565.613,A -85,B 0,C 180,E1 -26851.266,E2 -26851.266} C_VEL
LIN {X 0,Y 144.56,Z 564.569,A -85,B 0,C 180,E1 -26851.63,E2 -26851.63} C_VEL
LIN {X 0,Y 144.436,Z 565.495,A -85,B 0,C 180,E1 -26852.03,E2 -26852.03} C_VEL
LIN {X 0,Y 137.793,Z 576.825,A -85,B 0,C 180,E1 -26854.52,E2 -26854.52} C_VEL
LIN {X 0,Y 130.562,Z 587.138,A -85,B 0,C 180,E1 -26857.434,E2 -26857.434} C_VEL
LIN {X 0,Y 123.271,Z 596.279,A -85,B 0,C 180,E1 -26860.932,E2 -26860.932} C_VEL
LIN {X 0,Y 115.407,Z 605.008,A -85,B 0,C 180,E1 -26865.541,E2 -26865.541} C_VEL
LIN {X 0,Y 109.356,Z 611.156,A -85,B 0,C 180,E1 -26870.002,E2 -26870.002} C_VEL
LIN {X 0,Y 104.13,Z 616.238,A -85,B 0,C 180,E1 -26874.986,E2 -26874.986} C_VEL
LIN {X 0,Y 98.244,Z 621.496,A -85,B 0,C 180,E1 -26882.284,E2 -26882.284} C_VEL
LIN {X 0,Y 94.903,Z 624.43,A -85,B 0,C 180,E1 -26888.261,E2 -26888.261} C_VEL
LIN {X 0,Y 92.106,Z 627.123,A -85,B 0,C 180,E1 -26896.761,E2 -26896.761} C_VEL
LIN {X 0,Y 90.893,Z 628.467,A -85,B 0,C 180,E1 -26905.559,E2 -26905.559} C_VEL
LIN {X 0,Y 90.914,Z 628.642,A -85,B 0,C 180,E1 -26909.993,E2 -26909.993} C_VEL
LIN {X 0,Y 91.31,Z 628.009,A -85,B 0,C 180,E1 -26918.848,E2 -26918.848} C_VEL
LIN {X 0,Y 93.274,Z 626.042,A -85,B 0,C 180,E1 -26927.534,E2 -26927.534} C_VEL
LIN {X 0,Y 96.948,Z 622.689,A -85,B 0,C 180,E1 -26935.775,E2 -26935.775} C_VEL
LIN {X 0,Y 102.42,Z 617.847,A -85,B 0,C 180,E1 -26943.288,E2 -26943.288} C_VEL
LIN {X 0,Y 107.526,Z 613.072,A -85,B 0,C 180,E1 -26948.517,E2 -26948.517} C_VEL
LIN {X 0,Y 114.28,Z 606.391,A -85,B 0,C 180,E1 -26953.769,E2 -26953.769} C_VEL
LIN {X 0,Y 122.044,Z 597.956,A -85,B 0,C 180,E1 -26958.462,E2 -26958.462} C_VEL
LIN {X 0,Y 129.234,Z 589.153,A -85,B 0,C 180,E1 -26962.041,E2 -26962.041} C_VEL
LIN {X 0,Y 136.882,Z 578.483,A -85,B 0,C 180,E1 -26965.226,E2 -26965.226} C_VEL
LIN {X 0,Y 143.437,Z 567.69,A -85,B 0,C 180,E1 -26967.684,E2 -26967.684} C_VEL
LIN {X 0,Y 149.565,Z 555.879,A -85,B 0,C 180,E1 -26969.695,E2 -26969.695} C_VEL
LIN {X 0,Y 155.214,Z 542.824,A -85,B 0,C 180,E1 -26971.308,E2 -26971.308} C_VEL
LIN {X 0,Y 159.762,Z 529.389,A -85,B 0,C 180,E1 -26972.534,E2 -26972.534} C_VEL
LIN {X 0,Y 163.418,Z 514.772,A -85,B 0,C 180,E1 -26973.449,E2 -26973.449} C_VEL
LIN {X 0,Y 165.724,Z 500.683,A -85,B 0,C 180,E1 -26974.034,E2 -26974.034} C_VEL
LIN {X 0,Y 168.645,Z 471.213,A -85,B 0,C 180,E1 -26974.885,E2 -26974.885} C_VEL
LIN {X 0,Y 165.497,Z 464.044,A -85,B 0,C 180,E1 -26978.132,E2 -26978.132} C_VEL
LIN {X 0,Y 162.645,Z 458.221,A -85,B 0,C 180,E1 -26981.579,E2 -26981.579} C_VEL
LIN {X 0,Y 160.721,Z 454.646,A -85,B 0,C 180,E1 -26984.342,E2 -26984.342} C_VEL
LIN {X 0,Y 159.237,Z 451.817,A -85,B 0,C 180,E1 -26986.927,E2 -26986.927} C_VEL
LIN {X 0,Y 157.481,Z 448.317,A -85,B 0,C 180,E1 -26991.014,E2 -26991.014} C_VEL
LIN {X 0,Y 156.063,Z 444.277,A -85,B 0,C 180,E1 -27000,E2 -27000} C_VEL
LIN {X 0,Y 157.739,Z 448.853,A -85,B 0,C 180,E1 -27009.618,E2 -27009.618} C_VEL
LIN {X 0,Y 159.871,Z 453.035,A -85,B 0,C 180,E1 -27014.154,E2 -27014.154} C_VEL
LIN {X 0,Y 162.087,Z 457.171,A -85,B 0,C 180,E1 -27017.579,E2 -27017.579} C_VEL
LIN {X 0,Y 164.489,Z 461.962,A -85,B 0,C 180,E1 -27020.635,E2 -27020.635} C_VEL
LIN {X 0,Y 167.135,Z 467.852,A -85,B 0,C 180,E1 -27023.545,E2 -27023.545} C_VEL
LIN {X 0,Y 168.578,Z 472.308,A -85,B 0,C 180,E1 -27025.086,E2 -27025.086} C_VEL
LIN {X 0,Y 165.065,Z 505.988,A -85,B 0,C 180,E1 -27026.042,E2 -27026.042} C_VEL
LIN {X 0,Y 162.381,Z 520.379,A -85,B 0,C 180,E1 -27026.751,E2 -27026.751} C_VEL
LIN {X 0,Y 158.637,Z 533.785,A -85,B 0,C 180,E1 -27027.629,E2 -27027.629} C_VEL
LIN {X 0,Y 153.603,Z 547.65,A -85,B 0,C 180,E1 -27028.959,E2 -27028.959} C_VEL
LIN {X 0,Y 147.966,Z 560.062,A -85,B 0,C 180,E1 -27030.592,E2 -27030.592} C_VEL
LIN {X 0,Y 141.762,Z 571.406,A -85,B 0,C 180,E1 -27032.573,E2 -27032.573} C_VEL
LIN {X 0,Y 134.644,Z 582.698,A -85,B 0,C 180,E1 -27035.285,E2 -27035.285} C_VEL
LIN {X 0,Y 127.614,Z 592.224,A -85,B 0,C 180,E1 -27038.308,E2 -27038.308} C_VEL
LIN {X 0,Y 120.414,Z 600.789,A -85,B 0,C 180,E1 -27041.922,E2 -27041.922} C_VEL
LIN {X 0,Y 112.795,Z 608.987,A -85,B 0,C 180,E1 -27046.742,E2 -27046.742} C_VEL
LIN {X 0,Y 106.966,Z 614.733,A -85,B 0,C 180,E1 -27051.386,E2 -27051.386} C_VEL
LIN {X 0,Y 102.022,Z 619.438,A -85,B 0,C 180,E1 -27056.565,E2 -27056.565} C_VEL
LIN {X 0,Y 96.617,Z 624.319,A -85,B 0,C 180,E1 -27064.13,E2 -27064.13} C_VEL
LIN {X 0,Y 92.941,Z 627.709,A -85,B 0,C 180,E1 -27072.401,E2 -27072.401} C_VEL
LIN {X 0,Y 91.134,Z 629.71,A -85,B 0,C 180,E1 -27081.134,E2 -27081.134} C_VEL
LIN {X 0,Y 90.84,Z 630.365,A -85,B 0,C 180,E1 -27090.007,E2 -27090.007} C_VEL
LIN {X 0,Y 91.139,Z 629.677,A -85,B 0,C 180,E1 -27098.879,E2 -27098.879} C_VEL
LIN {X 0,Y 92.948,Z 627.645,A -85,B 0,C 180,E1 -27107.611,E2 -27107.611} C_VEL
LIN {X 0,Y 96.624,Z 624.227,A -85,B 0,C 180,E1 -27115.882,E2 -27115.882} C_VEL
LIN {X 0,Y 101.21,Z 620.092,A -85,B 0,C 180,E1 -27122.449,E2 -27122.449} C_VEL
LIN {X 0,Y 103.083,Z 617.926,A -85,B 0,C 180,E1 -27125.341,E2 -27125.341} C_VEL
LIN {X 0,Y 105.103,Z 613.97,A -85,B 0,C 180,E1 -27130.247,E2 -27130.247} C_VEL
LIN {X 0,Y 107.927,Z 609.559,A -85,B 0,C 180,E1 -27134.727,E2 -27134.727} C_VEL
LIN {X 0,Y 110.887,Z 606.51,A -85,B 0,C 180,E1 -27136.842,E2 -27136.842} C_VEL
LIN {X 0,Y 112.041,Z 605.503,A -85,B 0,C 180,E1 -27137.401,E2 -27137.401} C_VEL
LIN {X 0,Y 111.346,Z 604.453,A -85,B 0,C 180,E1 -27138.99,E2 -27138.99} C_VEL
LIN {X 0,Y 108.562,Z 604.18,A -85,B 0,C 180,E1 -27140.981,E2 -27140.981} C_VEL
LIN {X 0,Y 99.722,Z 602.315,A -85,B 0,C 180,E1 -27150.44,E2 -27150.44} C_VEL
LIN {X 0,Y 94.256,Z 598.248,A -85,B 0,C 180,E1 -27167.075,E2 -27167.075} C_VEL
LIN {X 0,Y 103.45,Z 589.928,A -85,B 0,C 180,E1 -27191.76,E2 -27191.76} C_VEL
LIN {X 0,Y 114.624,Z 584.627,A -85,B 0,C 180,E1 -27201.585,E2 -27201.585} C_VEL
LIN {X 0,Y 121.405,Z 581.693,A -85,B 0,C 180,E1 -27205.733,E2 -27205.733} C_VEL
LIN {X 0,Y 129.789,Z 577.193,A -85,B 0,C 180,E1 -27209.166,E2 -27209.166} C_VEL
LIN {X 0,Y 135.212,Z 574.53,A -85,B 0,C 180,E1 -27211.318,E2 -27211.318} C_VEL
LIN {X 0,Y 134.244,Z 576.377,A -85,B 0,C 180,E1 -27211.888,E2 -27211.888} C_VEL
LIN {X 0,Y 126.365,Z 587.208,A -85,B 0,C 180,E1 -27214.873,E2 -27214.873} C_VEL
LIN {X 0,Y 118.707,Z 596.349,A -85,B 0,C 180,E1 -27218.322,E2 -27218.322} C_VEL
LIN {X 0,Y 110.439,Z 605.077,A -85,B 0,C 180,E1 -27222.953,E2 -27222.953} C_VEL
LIN {X 0,Y 103.99,Z 611.225,A -85,B 0,C 180,E1 -27227.474,E2 -27227.474} C_VEL
LIN {X 0,Y 98.378,Z 616.307,A -85,B 0,C 180,E1 -27232.603,E2 -27232.603} C_VEL
LIN {X 0,Y 92.007,Z 621.564,A -85,B 0,C 180,E1 -27240.224,E2 -27240.224} C_VEL
LIN {X 0,Y 88.308,Z 624.499,A -85,B 0,C 180,E1 -27246.544,E2 -27246.544} C_VEL
LIN {X 0,Y 85.203,Z 627.191,A -85,B 0,C 180,E1 -27255.666,E2 -27255.666} C_VEL
LIN {X 0,Y 83.813,Z 628.535,A -85,B 0,C 180,E1 -27265.183,E2 -27265.183} C_VEL
LIN {X 0,Y 83.813,Z 628.71,A -85,B 0,C 180,E1 -27269.993,E2 -27269.993} C_VEL
LIN {X 0,Y 84.293,Z 628.076,A -85,B 0,C 180,E1 -27279.592,E2 -27279.592} C_VEL
LIN {X 0,Y 86.49,Z 626.109,A -85,B 0,C 180,E1 -27288.96,E2 -27288.96} C_VEL
LIN {X 0,Y 90.592,Z 622.755,A -85,B 0,C 180,E1 -27297.733,E2 -27297.733} C_VEL
LIN {X 0,Y 96.535,Z 617.913,A -85,B 0,C 180,E1 -27305.613,E2 -27305.613} C_VEL
LIN {X 0,Y 101.723,Z 613.424,A -85,B 0,C 180,E1 -27310.752,E2 -27310.752} C_VEL
LIN {X 0,Y 109.251,Z 606.457,A -85,B 0,C 180,E1 -27316.352,E2 -27316.352} C_VEL
LIN {X 0,Y 117.438,Z 598.021,A -85,B 0,C 180,E1 -27321.066,E2 -27321.066} C_VEL
LIN {X 0,Y 124.994,Z 589.218,A -85,B 0,C 180,E1 -27324.606,E2 -27324.606} C_VEL
LIN {X 0,Y 132.955,Z 578.547,A -85,B 0,C 180,E1 -27327.744,E2 -27327.744} C_VEL
LIN {X 0,Y 139.763,Z 567.754,A -85,B 0,C 180,E1 -27330.15,E2 -27330.15} C_VEL
LIN {X 0,Y 146.118,Z 555.942,A -85,B 0,C 180,E1 -27332.094,E2 -27332.094} C_VEL
LIN {X 0,Y 151.932,Z 542.885,A -85,B 0,C 180,E1 -27333.658,E2 -27333.658} C_VEL
LIN {X 0,Y 156.544,Z 529.676,A -85,B 0,C 180,E1 -27334.825,E2 -27334.825} C_VEL
LIN {X 0,Y 160.306,Z 515.151,A -85,B 0,C 180,E1 -27335.702,E2 -27335.702} C_VEL
LIN {X 0,Y 162.659,Z 501.436,A -85,B 0,C 180,E1 -27336.257,E2 -27336.257} C_VEL
LIN {X 0,Y 165.395,Z 474.699,A -85,B 0,C 180,E1 -27337.028,E2 -27337.028} C_VEL
LIN {X 0,Y 162.345,Z 467.516,A -85,B 0,C 180,E1 -27340.643,E2 -27340.643} C_VEL
LIN {X 0,Y 159.758,Z 462.044,A -85,B 0,C 180,E1 -27344.367,E2 -27344.367} C_VEL
LIN {X 0,Y 157.836,Z 458.327,A -85,B 0,C 180,E1 -27347.871,E2 -27347.871} C_VEL
LIN {X 0,Y 156.364,Z 455.172,A -85,B 0,C 180,E1 -27351.654,E2 -27351.654} C_VEL
LIN {X 0,Y 155.18,Z 451.471,A -85,B 0,C 180,E1 -27360,E2 -27360} C_VEL
LIN {X 0,Y 156.623,Z 455.703,A -85,B 0,C 180,E1 -27369.037,E2 -27369.037} C_VEL
LIN {X 0,Y 158.596,Z 459.855,A -85,B 0,C 180,E1 -27373.555,E2 -27373.555} C_VEL
LIN {X 0,Y 160.604,Z 463.876,A -85,B 0,C 180,E1 -27376.87,E2 -27376.87} C_VEL
LIN {X 0,Y 163.299,Z 469.696,A -85,B 0,C 180,E1 -27380.471,E2 -27380.471} C_VEL
LIN {X 0,Y 164.927,Z 473.8,A -85,B 0,C 180,E1 -27382.396,E2 -27382.396} C_VEL
LIN {X 0,Y 165.381,Z 475.269,A -85,B 0,C 180,E1 -27382.935,E2 -27382.935} C_VEL
LIN {X 0,Y 162.014,Z 506.328,A -85,B 0,C 180,E1 -27383.805,E2 -27383.805} C_VEL
LIN {X 0,Y 159.235,Z 520.615,A -85,B 0,C 180,E1 -27384.483,E2 -27384.483} C_VEL
LIN {X 0,Y 155.468,Z 533.724,A -85,B 0,C 180,E1 -27385.307,E2 -27385.307} C_VEL
LIN {X 0,Y 150.299,Z 547.589,A -85,B 0,C 180,E1 -27386.593,E2 -27386.593} C_VEL
LIN {X 0,Y 144.482,Z 559.999,A -85,B 0,C 180,E1 -27388.169,E2 -27388.169} C_VEL
LIN {X 0,Y 138.061,Z 571.342,A -85,B 0,C 180,E1 -27390.083,E2 -27390.083} C_VEL
LIN {X 0,Y 131.128,Z 581.951,A -85,B 0,C 180,E1 -27392.557,E2 -27392.557} C_VEL
LIN {X 0,Y 123.335,Z 592.159,A -85,B 0,C 180,E1 -27395.717,E2 -27395.717} C_VEL
LIN {X 0,Y 115.771,Z 600.724,A -85,B 0,C 180,E1 -27399.294,E2 -27399.294} C_VEL
LIN {X 0,Y 107.692,Z 608.921,A -85,B 0,C 180,E1 -27404.13,E2 -27404.13} C_VEL
LIN {X 0,Y 101.473,Z 614.667,A -85,B 0,C 180,E1 -27408.863,E2 -27408.863} C_VEL
LIN {X 0,Y 94.509,Z 620.759,A -85,B 0,C 180,E1 -27416.11,E2 -27416.11} C_VEL
LIN {X 0,Y 90.247,Z 624.252,A -85,B 0,C 180,E1 -27422.152,E2 -27422.152} C_VEL
LIN {X 0,Y 86.175,Z 627.642,A -85,B 0,C 180,E1 -27430.968,E2 -27430.968} C_VEL
LIN {X 0,Y 84.12,Z 629.643,A -85,B 0,C 180,E1 -27440.389,E2 -27440.389} C_VEL
LIN {X 0,Y 83.761,Z 630.298,A -85,B 0,C 180,E1 -27450.007,E2 -27450.007} C_VEL
LIN {X 0,Y 84.125,Z 629.609,A -85,B 0,C 180,E1 -27459.626,E2 -27459.626} C_VEL
LIN {X 0,Y 86.182,Z 627.577,A -85,B 0,C 180,E1 -27469.045,E2 -27469.045} C_VEL
LIN {X 0,Y 90.254,Z 624.159,A -85,B 0,C 180,E1 -27477.861,E2 -27477.861} C_VEL
LIN {X 0,Y 96.165,Z 619.252,A -85,B 0,C 180,E1 -27485.787,E2 -27485.787} C_VEL
LIN {X 0,Y 101.732,Z 614.518,A -85,B 0,C 180,E1 -27491.025,E2 -27491.025} C_VEL
LIN {X 0,Y 109.613,Z 607.662,A -85,B 0,C 180,E1 -27496.17,E2 -27496.17} C_VEL
LIN {X 0,Y 110.887,Z 606.51,A -85,B 0,C 180,E1 -27496.842,E2 -27496.842} C_VEL
LIN {X 0,Y 111.447,Z 605.607,A -85,B 0,C 180,E1 -27497.601,E2 -27497.601} C_VEL
LIN {X 0,Y 110.794,Z 604.664,A -85,B 0,C 180,E1 -27499.101,E2 -27499.101} C_VEL
LIN {X 0,Y 109.214,Z 604.315,A -85,B 0,C 180,E1 -27500.481,E2 -27500.481} C_VEL
LIN {X 0,Y 106.817,Z 604.298,A -85,B 0,C 180,E1 -27502.038,E2 -27502.038} C_VEL
LIN {X 0,Y 96.509,Z 605.807,A -85,B 0,C 180,E1 -27507.753,E2 -27507.753} C_VEL
LIN {X 0,Y 93.774,Z 605.892,A -85,B 0,C 180,E1 -27510.248,E2 -27510.248} C_VEL
LIN {X 0,Y 92.811,Z 605.702,A -85,B 0,C 180,E1 -27511.643,E2 -27511.643} C_VEL
LIN {X 0,Y 88.503,Z 602.593,A -85,B 0,C 180,E1 -27526.218,E2 -27526.218} C_VEL
LIN {X 0,Y 97.977,Z 594.798,A -85,B 0,C 180,E1 -27552.427,E2 -27552.427} C_VEL
LIN {X 0,Y 109.531,Z 589.896,A -85,B 0,C 180,E1 -27562.643,E2 -27562.643} C_VEL
LIN {X 0,Y 119.135,Z 586.062,A -85,B 0,C 180,E1 -27568.16,E2 -27568.16} C_VEL
LIN {X 0,Y 124.967,Z 583.212,A -85,B 0,C 180,E1 -27570.408,E2 -27570.408} C_VEL
LIN {X 0,Y 124.892,Z 584.2,A -85,B 0,C 180,E1 -27571.237,E2 -27571.237} C_VEL
LIN {X 0,Y 117.021,Z 593.544,A -85,B 0,C 180,E1 -27574.323,E2 -27574.323} C_VEL
LIN {X 0,Y 109.376,Z 601.626,A -85,B 0,C 180,E1 -27578.074,E2 -27578.074} C_VEL
LIN {X 0,Y 101.054,Z 609.366,A -85,B 0,C 180,E1 -27583.085,E2 -27583.085} C_VEL
LIN {X 0,Y 94.72,Z 614.77,A -85,B 0,C 180,E1 -27588.096,E2 -27588.096} C_VEL
LIN {X 0,Y 87.498,Z 620.446,A -85,B 0,C 180,E1 -27595.78,E2 -27595.78} C_VEL
LIN {X 0,Y 81.808,Z 624.567,A -85,B 0,C 180,E1 -27604.553,E2 -27604.553} C_VEL
LIN {X 0,Y 78.312,Z 627.259,A -85,B 0,C 180,E1 -27614.374,E2 -27614.374} C_VEL
LIN {X 0,Y 76.754,Z 628.602,A -85,B 0,C 180,E1 -27624.738,E2 -27624.738} C_VEL
LIN {X 0,Y 76.735,Z 628.777,A -85,B 0,C 180,E1 -27629.992,E2 -27629.992} C_VEL
LIN {X 0,Y 77.287,Z 628.143,A -85,B 0,C 180,E1 -27640.47,E2 -27640.47} C_VEL
LIN {X 0,Y 79.772,Z 626.176,A -85,B 0,C 180,E1 -27650.626,E2 -27650.626} C_VEL
LIN {X 0,Y 84.364,Z 622.822,A -85,B 0,C 180,E1 -27659.981,E2 -27659.981} C_VEL
LIN {X 0,Y 90.833,Z 617.98,A -85,B 0,C 180,E1 -27668.233,E2 -27668.233} C_VEL
LIN {X 0,Y 98.759,Z 611.507,A -85,B 0,C 180,E1 -27675.358,E2 -27675.358} C_VEL
LIN {X 0,Y 106.844,Z 604.296,A -85,B 0,C 180,E1 -27680.604,E2 -27680.604} C_VEL
LIN {X 0,Y 115.654,Z 595.37,A -85,B 0,C 180,E1 -27685.11,E2 -27685.11} C_VEL
LIN {X 0,Y 123.753,Z 585.991,A -85,B 0,C 180,E1 -27688.404,E2 -27688.404} C_VEL
LIN {X 0,Y 130.868,Z 576.349,A -85,B 0,C 180,E1 -27690.998,E2 -27690.998} C_VEL
LIN {X 0,Y 137.805,Z 565.433,A -85,B 0,C 180,E1 -27693.177,E2 -27693.177} C_VEL
LIN {X 0,Y 143.669,Z 554.573,A -85,B 0,C 180,E1 -27694.809,E2 -27694.809} C_VEL
LIN {X 0,Y 148.913,Z 542.947,A -85,B 0,C 180,E1 -27696.11,E2 -27696.11} C_VEL
LIN {X 0,Y 153.296,Z 530.871,A -85,B 0,C 180,E1 -27697.127,E2 -27697.127} C_VEL
LIN {X 0,Y 157.107,Z 517.109,A -85,B 0,C 180,E1 -27697.968,E2 -27697.968} C_VEL
LIN {X 0,Y 159.799,Z 502.54,A -85,B 0,C 180,E1 -27698.556,E2 -27698.556} C_VEL
LIN {X 0,Y 162.374,Z 478.288,A -85,B 0,C 180,E1 -27699.251,E2 -27699.251} C_VEL
LIN {X 0,Y 159.518,Z 471.287,A -85,B 0,C 180,E1 -27703.202,E2 -27703.202} C_VEL
LIN {X 0,Y 157.627,Z 467.321,A -85,B 0,C 180,E1 -27706.396,E2 -27706.396} C_VEL
LIN {X 0,Y 156.482,Z 464.808,A -85,B 0,C 180,E1 -27708.832,E2 -27708.832} C_VEL
LIN {X 0,Y 155.301,Z 462.064,A -85,B 0,C 180,E1 -27712.197,E2 -27712.197} C_VEL
LIN {X 0,Y 154.305,Z 458.592,A -85,B 0,C 180,E1 -27720,E2 -27720} C_VEL
LIN {X 0,Y 155.548,Z 462.611,A -85,B 0,C 180,E1 -27728.526,E2 -27728.526} C_VEL
LIN {X 0,Y 157.281,Z 466.549,A -85,B 0,C 180,E1 -27732.828,E2 -27732.828} C_VEL
LIN {X 0,Y 159.174,Z 470.642,A -85,B 0,C 180,E1 -27736.192,E2 -27736.192} C_VEL
LIN {X 0,Y 161.557,Z 476.263,A -85,B 0,C 180,E1 -27739.62,E2 -27739.62} C_VEL
LIN {X 0,Y 162.412,Z 478.493,A -85,B 0,C 180,E1 -27740.721,E2 -27740.721} C_VEL
LIN {X 0,Y 159.257,Z 506.462,A -85,B 0,C 180,E1 -27741.481,E2 -27741.481} C_VEL
LIN {X 0,Y 156.298,Z 521.057,A -85,B 0,C 180,E1 -27742.141,E2 -27742.141} C_VEL
LIN {X 0,Y 152.196,Z 534.795,A -85,B 0,C 180,E1 -27742.989,E2 -27742.989} C_VEL
LIN {X 0,Y 147.258,Z 547.527,A -85,B 0,C 180,E1 -27744.123,E2 -27744.123} C_VEL
LIN {X 0,Y 141.267,Z 559.936,A -85,B 0,C 180,E1 -27745.627,E2 -27745.627} C_VEL
LIN {X 0,Y 134.629,Z 571.279,A -85,B 0,C 180,E1 -27747.457,E2 -27747.457} C_VEL
LIN {X 0,Y 126.973,Z 582.542,A -85,B 0,C 180,E1 -27750.026,E2 -27750.026} C_VEL
LIN {X 0,Y 119.327,Z 592.094,A -85,B 0,C 180,E1 -27752.946,E2 -27752.946} C_VEL
LIN {X 0,Y 111.395,Z 600.659,A -85,B 0,C 180,E1 -27756.457,E2 -27756.457} C_VEL
LIN {X 0,Y 102.855,Z 608.855,A -85,B 0,C 180,E1 -27761.279,E2 -27761.279} C_VEL
LIN {X 0,Y 96.207,Z 614.601,A -85,B 0,C 180,E1 -27766.063,E2 -27766.063} C_VEL
LIN {X 0,Y 90.412,Z 619.304,A -85,B 0,C 180,E1 -27771.557,E2 -27771.557} C_VEL
LIN {X 0,Y 84.006,Z 624.185,A -85,B 0,C 180,E1 -27779.879,E2 -27779.879} C_VEL
LIN {X 0,Y 79.459,Z 627.575,A -85,B 0,C 180,E1 -27789.289,E2 -27789.289} C_VEL
LIN {X 0,Y 77.108,Z 629.576,A -85,B 0,C 180,E1 -27799.505,E2 -27799.505} C_VEL
LIN {X 0,Y 76.673,Z 630.231,A -85,B 0,C 180,E1 -27810.008,E2 -27810.008} C_VEL
LIN {X 0,Y 77.113,Z 629.542,A -85,B 0,C 180,E1 -27820.51,E2 -27820.51} C_VEL
LIN {X 0,Y 79.466,Z 627.509,A -85,B 0,C 180,E1 -27830.725,E2 -27830.725} C_VEL
LIN {X 0,Y 84.013,Z 624.091,A -85,B 0,C 180,E1 -27840.135,E2 -27840.135} C_VEL
LIN {X 0,Y 90.449,Z 619.183,A -85,B 0,C 180,E1 -27848.442,E2 -27848.442} C_VEL
LIN {X 0,Y 96.482,Z 614.449,A -85,B 0,C 180,E1 -27853.797,E2 -27853.797} C_VEL
LIN {X 0,Y 103.537,Z 608.688,A -85,B 0,C 180,E1 -27858.311,E2 -27858.311} C_VEL
LIN {X 0,Y 101.23,Z 607.563,A -85,B 0,C 180,E1 -27861.33,E2 -27861.33} C_VEL
LIN {X 0,Y 92.811,Z 605.702,A -85,B 0,C 180,E1 -27871.643,E2 -27871.643} C_VEL
LIN {X 0,Y 90.577,Z 605.357,A -85,B 0,C 180,E1 -27875.057,E2 -27875.057} C_VEL
LIN {X 0,Y 83.567,Z 605.881,A -85,B 0,C 180,E1 -27885.855,E2 -27885.855} C_VEL
LIN {X 0,Y 82.753,Z 605.553,A -85,B 0,C 180,E1 -27889.853,E2 -27889.853} C_VEL
LIN {X 0,Y 82.82,Z 605.289,A -85,B 0,C 180,E1 -27891.193,E2 -27891.193} C_VEL
LIN {X 0,Y 95.84,Z 597.954,A -85,B 0,C 180,E1 -27917.057,E2 -27917.057} C_VEL
LIN {X 0,Y 111.761,Z 592.186,A -85,B 0,C 180,E1 -27928.301,E2 -27928.301} C_VEL
LIN {X 0,Y 115.01,Z 591.015,A -85,B 0,C 180,E1 -27929.886,E2 -27929.886} C_VEL
LIN {X 0,Y 114.553,Z 592.13,A -85,B 0,C 180,E1 -27930.795,E2 -27930.795} C_VEL
LIN {X 0,Y 106.437,Z 600.467,A -85,B 0,C 180,E1 -27934.365,E2 -27934.365} C_VEL
LIN {X 0,Y 97.533,Z 608.43,A -85,B 0,C 180,E1 -27939.22,E2 -27939.22} C_VEL
LIN {X 0,Y 89.536,Z 614.839,A -85,B 0,C 180,E1 -27945.045,E2 -27945.045} C_VEL
LIN {X 0,Y 81.712,Z 620.515,A -85,B 0,C 180,E1 -27952.973,E2 -27952.973} C_VEL
LIN {X 0,Y 75.425,Z 624.635,A -85,B 0,C 180,E1 -27962.223,E2 -27962.223} C_VEL
LIN {X 0,Y 71.479,Z 627.327,A -85,B 0,C 180,E1 -27972.836,E2 -27972.836} C_VEL
LIN {X 0,Y 69.675,Z 628.67,A -85,B 0,C 180,E1 -27984.202,E2 -27984.202} C_VEL
LIN {X 0,Y 69.647,Z 628.844,A -85,B 0,C 180,E1 -27989.991,E2 -27989.991} C_VEL
LIN {X 0,Y 70.315,Z 628.21,A -85,B 0,C 180,E1 -28001.522,E2 -28001.522} C_VEL
LIN {X 0,Y 73.142,Z 626.243,A -85,B 0,C 180,E1 -28012.594,E2 -28012.594} C_VEL
LIN {X 0,Y 78.284,Z 622.888,A -85,B 0,C 180,E1 -28022.583,E2 -28022.583} C_VEL
LIN {X 0,Y 85.348,Z 618.046,A -85,B 0,C 180,E1 -28031.196,E2 -28031.196} C_VEL
LIN {X 0,Y 91.617,Z 613.377,A -85,B 0,C 180,E1 -28036.771,E2 -28036.771} C_VEL
LIN {X 0,Y 99.949,Z 606.589,A -85,B 0,C 180,E1 -28042.274,E2 -28042.274} C_VEL
LIN {X 0,Y 109.03,Z 598.152,A -85,B 0,C 180,E1 -28046.915,E2 -28046.915} C_VEL
LIN {X 0,Y 117.336,Z 589.347,A -85,B 0,C 180,E1 -28050.272,E2 -28050.272} C_VEL
LIN {X 0,Y 125.922,Z 578.676,A -85,B 0,C 180,E1 -28053.24,E2 -28053.24} C_VEL
LIN {X 0,Y 133.247,Z 567.881,A -85,B 0,C 180,E1 -28055.47,E2 -28055.47} C_VEL
LIN {X 0,Y 140.03,Z 556.067,A -85,B 0,C 180,E1 -28057.241,E2 -28057.241} C_VEL
LIN {X 0,Y 146.188,Z 543.008,A -85,B 0,C 180,E1 -28058.65,E2 -28058.65} C_VEL
LIN {X 0,Y 151.184,Z 529.38,A -85,B 0,C 180,E1 -28059.728,E2 -28059.728} C_VEL
LIN {X 0,Y 155.044,Z 515.103,A -85,B 0,C 180,E1 -28060.492,E2 -28060.492} C_VEL
LIN {X 0,Y 157.441,Z 501.852,A -85,B 0,C 180,E1 -28060.979,E2 -28060.979} C_VEL
LIN {X 0,Y 159.599,Z 482.112,A -85,B 0,C 180,E1 -28061.531,E2 -28061.531} C_VEL
LIN {X 0,Y 157.487,Z 476.772,A -85,B 0,C 180,E1 -28064.888,E2 -28064.888} C_VEL
LIN {X 0,Y 155.595,Z 472.168,A -85,B 0,C 180,E1 -28068.767,E2 -28068.767} C_VEL
LIN {X 0,Y 154.309,Z 469.025,A -85,B 0,C 180,E1 -28072.558,E2 -28072.558} C_VEL
LIN {X 0,Y 153.424,Z 465.765,A -85,B 0,C 180,E1 -28080,E2 -28080} C_VEL
LIN {X 0,Y 154.469,Z 469.477,A -85,B 0,C 180,E1 -28087.949,E2 -28087.949} C_VEL
LIN {X 0,Y 155.961,Z 473.205,A -85,B 0,C 180,E1 -28092.029,E2 -28092.029} C_VEL
LIN {X 0,Y 157.772,Z 477.363,A -85,B 0,C 180,E1 -28095.502,E2 -28095.502} C_VEL
LIN {X 0,Y 159.653,Z 482.297,A -85,B 0,C 180,E1 -28098.464,E2 -28098.464} C_VEL
LIN {X 0,Y 156.742,Z 506.745,A -85,B 0,C 180,E1 -28099.08,E2 -28099.08} C_VEL
LIN {X 0,Y 153.622,Z 521.545,A -85,B 0,C 180,E1 -28099.716,E2 -28099.716} C_VEL
LIN {X 0,Y 149.558,Z 534.734,A -85,B 0,C 180,E1 -28100.477,E2 -28100.477} C_VEL
LIN {X 0,Y 144.505,Z 547.465,A -85,B 0,C 180,E1 -28101.556,E2 -28101.556} C_VEL
LIN {X 0,Y 138.339,Z 559.873,A -85,B 0,C 180,E1 -28102.969,E2 -28102.969} C_VEL
LIN {X 0,Y 131.508,Z 571.215,A -85,B 0,C 180,E1 -28104.712,E2 -28104.712} C_VEL
LIN {X 0,Y 123.566,Z 582.477,A -85,B 0,C 180,E1 -28107.168,E2 -28107.168} C_VEL
LIN {X 0,Y 115.615,Z 592.029,A -85,B 0,C 180,E1 -28109.988,E2 -28109.988} C_VEL
LIN {X 0,Y 107.318,Z 600.593,A -85,B 0,C 180,E1 -28113.399,E2 -28113.399} C_VEL
LIN {X 0,Y 98.305,Z 608.789,A -85,B 0,C 180,E1 -28118.16,E2 -28118.16} C_VEL
LIN {X 0,Y 91.204,Z 614.535,A -85,B 0,C 180,E1 -28122.952,E2 -28122.952} C_VEL
LIN {X 0,Y 83.037,Z 620.626,A -85,B 0,C 180,E1 -28130.606,E2 -28130.606} C_VEL
LIN {X 0,Y 77.921,Z 624.118,A -85,B 0,C 180,E1 -28137.247,E2 -28137.247} C_VEL
LIN {X 0,Y 72.811,Z 627.508,A -85,B 0,C 180,E1 -28147.298,E2 -28147.298} C_VEL
LIN {X 0,Y 70.106,Z 629.508,A -85,B 0,C 180,E1 -28158.443,E2 -28158.443} C_VEL
LIN {X 0,Y 69.574,Z 630.163,A -85,B 0,C 180,E1 -28170.009,E2 -28170.009} C_VEL
LIN {X 0,Y 70.111,Z 629.474,A -85,B 0,C 180,E1 -28181.574,E2 -28181.574} C_VEL
LIN {X 0,Y 72.819,Z 627.441,A -85,B 0,C 180,E1 -28192.718,E2 -28192.718} C_VEL
LIN {X 0,Y 77.93,Z 624.022,A -85,B 0,C 180,E1 -28202.767,E2 -28202.767} C_VEL
LIN {X 0,Y 84.954,Z 619.114,A -85,B 0,C 180,E1 -28211.447,E2 -28211.447} C_VEL
LIN {X 0,Y 91.478,Z 614.381,A -85,B 0,C 180,E1 -28216.883,E2 -28216.883} C_VEL
LIN {X 0,Y 95.207,Z 611.562,A -85,B 0,C 180,E1 -28219.31,E2 -28219.31} C_VEL
LIN {X 0,Y 94.303,Z 610.842,A -85,B 0,C 180,E1 -28221.107,E2 -28221.107} C_VEL
LIN {X 0,Y 86.766,Z 609.282,A -85,B 0,C 180,E1 -28230.923,E2 -28230.923} C_VEL
LIN {X 0,Y 82.61,Z 606.622,A -85,B 0,C 180,E1 -28245.214,E2 -28245.214} C_VEL
LIN {X 0,Y 82.82,Z 605.289,A -85,B 0,C 180,E1 -28251.193,E2 -28251.193} C_VEL
LIN {X 0,Y 82.962,Z 604.703,A -85,B 0,C 180,E1 -28255.255,E2 -28255.255} C_VEL
LIN {X 0,Y 82.607,Z 604.691,A -85,B 0,C 180,E1 -28262.12,E2 -28262.12} C_VEL
LIN {X 0,Y 83.081,Z 604.738,A -85,B 0,C 180,E1 -28267.609,E2 -28267.609} C_VEL
LIN {X 0,Y 84.575,Z 604.347,A -85,B 0,C 180,E1 -28271.508,E2 -28271.508} C_VEL
LIN {X 0,Y 85.366,Z 604.055,A -85,B 0,C 180,E1 -28272.711,E2 -28272.711} C_VEL
LIN {X 0,Y 98.894,Z 599.49,A -85,B 0,C 180,E1 -28285.239,E2 -28285.239} C_VEL
LIN {X 0,Y 103.865,Z 597.863,A -85,B 0,C 180,E1 -28288.272,E2 -28288.272} C_VEL
LIN {X 0,Y 105.377,Z 597.909,A -85,B 0,C 180,E1 -28289.875,E2 -28289.875} C_VEL
LIN {X 0,Y 95.824,Z 606.398,A -85,B 0,C 180,E1 -28294.39,E2 -28294.39} C_VEL
LIN {X 0,Y 86.974,Z 613.236,A -85,B 0,C 180,E1 -28299.846,E2 -28299.846} C_VEL
LIN {X 0,Y 80.21,Z 617.95,A -85,B 0,C 180,E1 -28305.486,E2 -28305.486} C_VEL
LIN {X 0,Y 72.431,Z 622.829,A -85,B 0,C 180,E1 -28314.386,E2 -28314.386} C_VEL
LIN {X 0,Y 66.645,Z 626.222,A -85,B 0,C 180,E1 -28325.041,E2 -28325.041} C_VEL
LIN {X 0,Y 63.367,Z 628.232,A -85,B 0,C 180,E1 -28337.174,E2 -28337.174} C_VEL
LIN {X 0,Y 62.548,Z 628.911,A -85,B 0,C 180,E1 -28349.99,E2 -28349.99} C_VEL
LIN {X 0,Y 63.356,Z 628.278,A -85,B 0,C 180,E1 -28362.808,E2 -28362.808} C_VEL
LIN {X 0,Y 66.622,Z 626.31,A -85,B 0,C 180,E1 -28374.948,E2 -28374.948} C_VEL
LIN {X 0,Y 72.393,Z 622.955,A -85,B 0,C 180,E1 -28385.615,E2 -28385.615} C_VEL
LIN {X 0,Y 80.122,Z 618.113,A -85,B 0,C 180,E1 -28394.555,E2 -28394.555} C_VEL
LIN {X 0,Y 86.893,Z 613.443,A -85,B 0,C 180,E1 -28400.196,E2 -28400.196} C_VEL
LIN {X 0,Y 95.761,Z 606.654,A -85,B 0,C 180,E1 -28405.642,E2 -28405.642} C_VEL
LIN {X 0,Y 105.303,Z 598.218,A -85,B 0,C 180,E1 -28410.171,E2 -28410.171} C_VEL
LIN {X 0,Y 113.974,Z 589.412,A -85,B 0,C 180,E1 -28413.381,E2 -28413.381} C_VEL
LIN {X 0,Y 121.394,Z 580.689,A -85,B 0,C 180,E1 -28415.746,E2 -28415.746} C_VEL
LIN {X 0,Y 128.93,Z 570.289,A -85,B 0,C 180,E1 -28417.908,E2 -28417.908} C_VEL
LIN {X 0,Y 135.872,Z 558.978,A -85,B 0,C 180,E1 -28419.624,E2 -28419.624} C_VEL
LIN {X 0,Y 142.183,Z 546.601,A -85,B 0,C 180,E1 -28420.953,E2 -28420.953} C_VEL
LIN {X 0,Y 147.739,Z 532.776,A -85,B 0,C 180,E1 -28422.05,E2 -28422.05} C_VEL
LIN {X 0,Y 151.924,Z 518.895,A -85,B 0,C 180,E1 -28422.831,E2 -28422.831} C_VEL
LIN {X 0,Y 154.878,Z 504.546,A -85,B 0,C 180,E1 -28423.393,E2 -28423.393} C_VEL
LIN {X 0,Y 157.048,Z 486.082,A -85,B 0,C 180,E1 -28423.911,E2 -28423.911} C_VEL
LIN {X 0,Y 155.321,Z 481.367,A -85,B 0,C 180,E1 -28427.236,E2 -28427.236} C_VEL
LIN {X 0,Y 153.974,Z 478.023,A -85,B 0,C 180,E1 -28430.586,E2 -28430.586} C_VEL
LIN {X 0,Y 153.214,Z 475.809,A -85,B 0,C 180,E1 -28433.332,E2 -28433.332} C_VEL
LIN {X 0,Y 152.55,Z 472.887,A -85,B 0,C 180,E1 -28440,E2 -28440} C_VEL
LIN {X 0,Y 153.378,Z 476.224,A -85,B 0,C 180,E1 -28447.239,E2 -28447.239} C_VEL
LIN {X 0,Y 154.667,Z 479.811,A -85,B 0,C 180,E1 -28451.197,E2 -28451.197} C_VEL
LIN {X 0,Y 156.28,Z 483.891,A -85,B 0,C 180,E1 -28454.606,E2 -28454.606} C_VEL
LIN {X 0,Y 157.118,Z 486.276,A -85,B 0,C 180,E1 -28456.121,E2 -28456.121} C_VEL
LIN {X 0,Y 154.466,Z 507.258,A -85,B 0,C 180,E1 -28456.609,E2 -28456.609} C_VEL
LIN {X 0,Y 151.314,Z 521.724,A -85,B 0,C 180,E1 -28457.199,E2 -28457.199} C_VEL
LIN {X 0,Y 147.226,Z 534.674,A -85,B 0,C 180,E1 -28457.888,E2 -28457.888} C_VEL
LIN {X 0,Y 142.05,Z 547.404,A -85,B 0,C 180,E1 -28458.891,E2 -28458.891} C_VEL
LIN {X 0,Y 135.723,Z 559.81,A -85,B 0,C 180,E1 -28460.206,E2 -28460.206} C_VEL
LIN {X 0,Y 128.701,Z 571.151,A -85,B 0,C 180,E1 -28461.839,E2 -28461.839} C_VEL
LIN {X 0,Y 120.986,Z 581.747,A -85,B 0,C 180,E1 -28463.993,E2 -28463.993} C_VEL
LIN {X 0,Y 112.23,Z 591.964,A -85,B 0,C 180,E1 -28466.843,E2 -28466.843} C_VEL
LIN {X 0,Y 103.557,Z 600.528,A -85,B 0,C 180,E1 -28470.097,E2 -28470.097} C_VEL
LIN {X 0,Y 94.062,Z 608.723,A -85,B 0,C 180,E1 -28474.738,E2 -28474.738} C_VEL
LIN {X 0,Y 86.499,Z 614.469,A -85,B 0,C 180,E1 -28479.49,E2 -28479.49} C_VEL
LIN {X 0,Y 79.683,Z 619.17,A -85,B 0,C 180,E1 -28485.134,E2 -28485.134} C_VEL
LIN {X 0,Y 72.028,Z 624.052,A -85,B 0,C 180,E1 -28494.177,E2 -28494.177} C_VEL
LIN {X 0,Y 66.271,Z 627.441,A -85,B 0,C 180,E1 -28504.911,E2 -28504.911} C_VEL
LIN {X 0,Y 63.146,Z 629.441,A -85,B 0,C 180,E1 -28517.148,E2 -28517.148} C_VEL
LIN {X 0,Y 62.492,Z 630.096,A -85,B 0,C 180,E1 -28530.01,E2 -28530.01} C_VEL
LIN {X 0,Y 63.152,Z 629.406,A -85,B 0,C 180,E1 -28542.87,E2 -28542.87} C_VEL
LIN {X 0,Y 66.28,Z 627.372,A -85,B 0,C 180,E1 -28555.106,E2 -28555.106} C_VEL
LIN {X 0,Y 72.038,Z 623.954,A -85,B 0,C 180,E1 -28565.838,E2 -28565.838} C_VEL
LIN {X 0,Y 79.735,Z 619.046,A -85,B 0,C 180,E1 -28574.851,E2 -28574.851} C_VEL
LIN {X 0,Y 85.95,Z 614.899,A -85,B 0,C 180,E1 -28579.77,E2 -28579.77} C_VEL
LIN {X 0,Y 86.65,Z 613.782,A -85,B 0,C 180,E1 -28581.463,E2 -28581.463} C_VEL
LIN {X 0,Y 79.966,Z 612.336,A -85,B 0,C 180,E1 -28591.521,E2 -28591.521} C_VEL
LIN {X 0,Y 76.536,Z 609.351,A -85,B 0,C 180,E1 -28609.418,E2 -28609.418} C_VEL
LIN {X 0,Y 85.366,Z 604.055,A -85,B 0,C 180,E1 -28632.711,E2 -28632.711} C_VEL
LIN {X 0,Y 86.709,Z 603.764,A -85,B 0,C 180,E1 -28635.207,E2 -28635.207} C_VEL
LIN {X 0,Y 89.774,Z 604.601,A -85,B 0,C 180,E1 -28643.732,E2 -28643.732} C_VEL
LIN {X 0,Y 91.878,Z 604.235,A -85,B 0,C 180,E1 -28645.842,E2 -28645.842} C_VEL
LIN {X 0,Y 96.219,Z 603.063,A -85,B 0,C 180,E1 -28648.765,E2 -28648.765} C_VEL
LIN {X 0,Y 87.845,Z 609.573,A -85,B 0,C 180,E1 -28652.843,E2 -28652.843} C_VEL
LIN {X 0,Y 78.292,Z 616.152,A -85,B 0,C 180,E1 -28659.178,E2 -28659.178} C_VEL
LIN {X 0,Y 70.826,Z 620.652,A -85,B 0,C 180,E1 -28665.993,E2 -28665.993} C_VEL
LIN {X 0,Y 63.155,Z 624.772,A -85,B 0,C 180,E1 -28676.181,E2 -28676.181} C_VEL
LIN {X 0,Y 58.018,Z 627.463,A -85,B 0,C 180,E1 -28688.68,E2 -28688.68} C_VEL
LIN {X 0,Y 55.565,Z 628.805,A -85,B 0,C 180,E1 -28702.723,E2 -28702.723} C_VEL
LIN {X 0,Y 55.466,Z 628.978,A -85,B 0,C 180,E1 -28709.989,E2 -28709.989} C_VEL
LIN {X 0,Y 56.449,Z 628.345,A -85,B 0,C 180,E1 -28724.407,E2 -28724.407} C_VEL
LIN {X 0,Y 60.245,Z 626.376,A -85,B 0,C 180,E1 -28737.804,E2 -28737.804} C_VEL
LIN {X 0,Y 66.717,Z 623.021,A -85,B 0,C 180,E1 -28749.189,E2 -28749.189} C_VEL
LIN {X 0,Y 75.207,Z 618.179,A -85,B 0,C 180,E1 -28758.369,E2 -28758.369} C_VEL
LIN {X 0,Y 82.511,Z 613.509,A -85,B 0,C 180,E1 -28764.002,E2 -28764.002} C_VEL
LIN {X 0,Y 91.931,Z 606.72,A -85,B 0,C 180,E1 -28769.308,E2 -28769.308} C_VEL
LIN {X 0,Y 101.944,Z 598.283,A -85,B 0,C 180,E1 -28773.651,E2 -28773.651} C_VEL
LIN {X 0,Y 110.965,Z 589.477,A -85,B 0,C 180,E1 -28776.672,E2 -28776.672} C_VEL
LIN {X 0,Y 118.646,Z 580.753,A -85,B 0,C 180,E1 -28778.883,E2 -28778.883} C_VEL
LIN {X 0,Y 126.423,Z 570.353,A -85,B 0,C 180,E1 -28780.901,E2 -28780.901} C_VEL
LIN {X 0,Y 133.568,Z 559.041,A -85,B 0,C 180,E1 -28782.477,E2 -28782.477} C_VEL
LIN {X 0,Y 140.026,Z 546.663,A -85,B 0,C 180,E1 -28783.7,E2 -28783.7} C_VEL
LIN {X 0,Y 145.704,Z 532.836,A -85,B 0,C 180,E1 -28784.712,E2 -28784.712} C_VEL
LIN {X 0,Y 150.013,Z 518.84,A -85,B 0,C 180,E1 -28785.426,E2 -28785.426} C_VEL
LIN {X 0,Y 153.046,Z 504.379,A -85,B 0,C 180,E1 -28785.938,E2 -28785.938} C_VEL
LIN {X 0,Y 154.8,Z 490.352,A -85,B 0,C 180,E1 -28786.271,E2 -28786.271} C_VEL
LIN {X 0,Y 153.377,Z 486.264,A -85,B 0,C 180,E1 -28789.661,E2 -28789.661} C_VEL
LIN {X 0,Y 152.164,Z 482.645,A -85,B 0,C 180,E1 -28794.035,E2 -28794.035} C_VEL
LIN {X 0,Y 151.674,Z 480.021,A -85,B 0,C 180,E1 -28800,E2 -28800} C_VEL
LIN {X 0,Y 152.331,Z 483.11,A -85,B 0,C 180,E1 -28806.644,E2 -28806.644} C_VEL
LIN {X 0,Y 153.557,Z 486.845,A -85,B 0,C 180,E1 -28810.757,E2 -28810.757} C_VEL
LIN {X 0,Y 154.817,Z 490.412,A -85,B 0,C 180,E1 -28813.678,E2 -28813.678} C_VEL
LIN {X 0,Y 152.334,Z 508.651,A -85,B 0,C 180,E1 -28814.102,E2 -28814.102} C_VEL
LIN {X 0,Y 148.994,Z 523.076,A -85,B 0,C 180,E1 -28814.664,E2 -28814.664} C_VEL
LIN {X 0,Y 144.39,Z 536.869,A -85,B 0,C 180,E1 -28815.364,E2 -28815.364} C_VEL
LIN {X 0,Y 139.096,Z 549.108,A -85,B 0,C 180,E1 -28816.278,E2 -28816.278} C_VEL
LIN {X 0,Y 132.637,Z 561.164,A -85,B 0,C 180,E1 -28817.51,E2 -28817.51} C_VEL
LIN {X 0,Y 124.638,Z 573.336,A -85,B 0,C 180,E1 -28819.198,E2 -28819.198} C_VEL
LIN {X 0,Y 116.101,Z 584.275,A -85,B 0,C 180,E1 -28821.448,E2 -28821.448} C_VEL
LIN {X 0,Y 107.662,Z 593.408,A -85,B 0,C 180,E1 -28823.966,E2 -28823.966} C_VEL
LIN {X 0,Y 98.721,Z 601.718,A -85,B 0,C 180,E1 -28827.156,E2 -28827.156} C_VEL
LIN {X 0,Y 88.801,Z 609.666,A -85,B 0,C 180,E1 -28831.716,E2 -28831.716} C_VEL
LIN {X 0,Y 79.601,Z 616.062,A -85,B 0,C 180,E1 -28837.395,E2 -28837.395} C_VEL
LIN {X 0,Y 70.376,Z 621.739,A -85,B 0,C 180,E1 -28845.663,E2 -28845.663} C_VEL
LIN {X 0,Y 62.802,Z 625.858,A -85,B 0,C 180,E1 -28855.988,E2 -28855.988} C_VEL
LIN {X 0,Y 57.708,Z 628.544,A -85,B 0,C 180,E1 -28868.582,E2 -28868.582} C_VEL
LIN {X 0,Y 55.458,Z 629.868,A -85,B 0,C 180,E1 -28882.731,E2 -28882.731} C_VEL
LIN {X 0,Y 55.393,Z 630.029,A -85,B 0,C 180,E1 -28890.011,E2 -28890.011} C_VEL
LIN {X 0,Y 56.244,Z 629.338,A -85,B 0,C 180,E1 -28904.483,E2 -28904.483} C_VEL
LIN {X 0,Y 59.884,Z 627.304,A -85,B 0,C 180,E1 -28918.009,E2 -28918.009} C_VEL
LIN {X 0,Y 66.388,Z 623.885,A -85,B 0,C 180,E1 -28929.444,E2 -28929.444} C_VEL
LIN {X 0,Y 74.833,Z 618.977,A -85,B 0,C 180,E1 -28938.717,E2 -28938.717} C_VEL
LIN {X 0,Y 77.246,Z 617.535,A -85,B 0,C 180,E1 -28940.663,E2 -28940.663} C_VEL
LIN {X 0,Y 78.144,Z 616.401,A -85,B 0,C 180,E1 -28942.729,E2 -28942.729} C_VEL
LIN {X 0,Y 71.596,Z 614.523,A -85,B 0,C 180,E1 -28956.881,E2 -28956.881} C_VEL
LIN {X 0,Y 70.743,Z 612.044,A -85,B 0,C 180,E1 -28973.51,E2 -28973.51} C_VEL
LIN {X 0,Y 84.224,Z 606.448,A -85,B 0,C 180,E1 -28999.499,E2 -28999.499} C_VEL
LIN {X 0,Y 91.878,Z 604.235,A -85,B 0,C 180,E1 -29005.842,E2 -29005.842} C_VEL
LIN {X 0,Y 92.184,Z 604.396,A -85,B 0,C 180,E1 -29006.6,E2 -29006.6} C_VEL
LIN {X 0,Y 91.286,Z 605.47,A -85,B 0,C 180,E1 -29007.832,E2 -29007.832} C_VEL
LIN {X 0,Y 88.814,Z 607.429,A -85,B 0,C 180,E1 -29009.096,E2 -29009.096} C_VEL
LIN {X 0,Y 78.517,Z 613.498,A -85,B 0,C 180,E1 -29012.072,E2 -29012.072} C_VEL
LIN {X 0,Y 76.602,Z 614.612,A -85,B 0,C 180,E1 -29013.096,E2 -29013.096} C_VEL
LIN {X 0,Y 68.259,Z 619.485,A -85,B 0,C 180,E1 -29019.435,E2 -29019.435} C_VEL
LIN {X 0,Y 61.399,Z 622.966,A -85,B 0,C 180,E1 -29026.611,E2 -29026.611} C_VEL
LIN {X 0,Y 54.062,Z 626.358,A -85,B 0,C 180,E1 -29038.655,E2 -29038.655} C_VEL
LIN {X 0,Y 49.595,Z 628.367,A -85,B 0,C 180,E1 -29053.523,E2 -29053.523} C_VEL
LIN {X 0,Y 48.368,Z 629.045,A -85,B 0,C 180,E1 -29069.987,E2 -29069.987} C_VEL
LIN {X 0,Y 49.584,Z 628.412,A -85,B 0,C 180,E1 -29086.455,E2 -29086.455} C_VEL
LIN {X 0,Y 54.039,Z 626.443,A -85,B 0,C 180,E1 -29101.333,E2 -29101.333} C_VEL
LIN {X 0,Y 61.354,Z 623.088,A -85,B 0,C 180,E1 -29113.402,E2 -29113.402} C_VEL
LIN {X 0,Y 70.672,Z 618.245,A -85,B 0,C 180,E1 -29122.694,E2 -29122.694} C_VEL
LIN {X 0,Y 78.532,Z 613.575,A -85,B 0,C 180,E1 -29128.215,E2 -29128.215} C_VEL
LIN {X 0,Y 88.493,Z 606.786,A -85,B 0,C 180,E1 -29133.294,E2 -29133.294} C_VEL
LIN {X 0,Y 98.987,Z 598.349,A -85,B 0,C 180,E1 -29137.349,E2 -29137.349} C_VEL
LIN {X 0,Y 108.346,Z 589.542,A -85,B 0,C 180,E1 -29140.127,E2 -29140.127} C_VEL
LIN {X 0,Y 117.072,Z 579.818,A -85,B 0,C 180,E1 -29142.381,E2 -29142.381} C_VEL
LIN {X 0,Y 125.902,Z 568.072,A -85,B 0,C 180,E1 -29144.328,E2 -29144.328} C_VEL
LIN {X 0,Y 133.243,Z 556.255,A -85,B 0,C 180,E1 -29145.722,E2 -29145.722} C_VEL
LIN {X 0,Y 139.852,Z 543.193,A -85,B 0,C 180,E1 -29146.797,E2 -29146.797} C_VEL
LIN {X 0,Y 145.247,Z 529.378,A -85,B 0,C 180,E1 -29147.639,E2 -29147.639} C_VEL
LIN {X 0,Y 149.412,Z 514.763,A -85,B 0,C 180,E1 -29148.219,E2 -29148.219} C_VEL
LIN {X 0,Y 151.935,Z 501.349,A -85,B 0,C 180,E1 -29148.604,E2 -29148.604} C_VEL
LIN {X 0,Y 152.754,Z 494.789,A -85,B 0,C 180,E1 -29148.787,E2 -29148.787} C_VEL
LIN {X 0,Y 151.719,Z 491.518,A -85,B 0,C 180,E1 -29152.012,E2 -29152.012} C_VEL
LIN {X 0,Y 151.154,Z 489.504,A -85,B 0,C 180,E1 -29154.664,E2 -29154.664} C_VEL
LIN {X 0,Y 150.796,Z 487.176,A -85,B 0,C 180,E1 -29160,E2 -29160} C_VEL
LIN {X 0,Y 151.291,Z 489.891,A -85,B 0,C 180,E1 -29165.957,E2 -29165.957} C_VEL
LIN {X 0,Y 152.344,Z 493.577,A -85,B 0,C 180,E1 -29169.998,E2 -29169.998} C_VEL
LIN {X 0,Y 152.769,Z 494.824,A -85,B 0,C 180,E1 -29171.161,E2 -29171.161} C_VEL
LIN {X 0,Y 150.435,Z 510.426,A -85,B 0,C 180,E1 -29171.547,E2 -29171.547} C_VEL
LIN {X 0,Y 146.795,Z 524.946,A -85,B 0,C 180,E1 -29172.069,E2 -29172.069} C_VEL
LIN {X 0,Y 142.263,Z 537.836,A -85,B 0,C 180,E1 -29172.685,E2 -29172.685} C_VEL
LIN {X 0,Y 136.447,Z 550.665,A -85,B 0,C 180,E1 -29173.564,E2 -29173.564} C_VEL
LIN {X 0,Y 129.852,Z 562.407,A -85,B 0,C 180,E1 -29174.68,E2 -29174.68} C_VEL
LIN {X 0,Y 122.487,Z 573.272,A -85,B 0,C 180,E1 -29176.059,E2 -29176.059} C_VEL
LIN {X 0,Y 114.805,Z 582.958,A -85,B 0,C 180,E1 -29177.823,E2 -29177.823} C_VEL
LIN {X 0,Y 104.971,Z 593.343,A -85,B 0,C 180,E1 -29180.412,E2 -29180.412} C_VEL
LIN {X 0,Y 95.67,Z 601.653,A -85,B 0,C 180,E1 -29183.344,E2 -29183.344} C_VEL
LIN {X 0,Y 85.268,Z 609.6,A -85,B 0,C 180,E1 -29187.637,E2 -29187.637} C_VEL
LIN {X 0,Y 75.477,Z 615.996,A -85,B 0,C 180,E1 -29193.083,E2 -29193.083} C_VEL
LIN {X 0,Y 65.462,Z 621.672,A -85,B 0,C 180,E1 -29201.292,E2 -29201.292} C_VEL
LIN {X 0,Y 57.041,Z 625.791,A -85,B 0,C 180,E1 -29211.986,E2 -29211.986} C_VEL
LIN {X 0,Y 51.121,Z 628.477,A -85,B 0,C 180,E1 -29225.655,E2 -29225.655} C_VEL
LIN {X 0,Y 48.41,Z 629.801,A -85,B 0,C 180,E1 -29241.665,E2 -29241.665} C_VEL
LIN {X 0,Y 48.309,Z 629.962,A -85,B 0,C 180,E1 -29250.013,E2 -29250.013} C_VEL
LIN {X 0,Y 49.368,Z 629.27,A -85,B 0,C 180,E1 -29266.555,E2 -29266.555} C_VEL
LIN {X 0,Y 53.68,Z 627.236,A -85,B 0,C 180,E1 -29281.593,E2 -29281.593} C_VEL
LIN {X 0,Y 61.025,Z 623.817,A -85,B 0,C 180,E1 -29293.722,E2 -29293.722} C_VEL
LIN {X 0,Y 70.44,Z 618.83,A -85,B 0,C 180,E1 -29303.228,E2 -29303.228} C_VEL
LIN {X 0,Y 63.786,Z 616.065,A -85,B 0,C 180,E1 -29327.27,E2 -29327.27} C_VEL
LIN {X 0,Y 78.238,Z 610.216,A -85,B 0,C 180,E1 -29361.059,E2 -29361.059} C_VEL
LIN {X 0,Y 85.6,Z 608.352,A -85,B 0,C 180,E1 -29367.285,E2 -29367.285} C_VEL
LIN {X 0,Y 84.758,Z 609.246,A -85,B 0,C 180,E1 -29368.487,E2 -29368.487} C_VEL
LIN {X 0,Y 76.602,Z 614.612,A -85,B 0,C 180,E1 -29373.096,E2 -29373.096} C_VEL
LIN {X 0,Y 72.174,Z 617.065,A -85,B 0,C 180,E1 -29375.465,E2 -29375.465} C_VEL
LIN {X 0,Y 60.46,Z 621.929,A -85,B 0,C 180,E1 -29380.452,E2 -29380.452} C_VEL
LIN {X 0,Y 54.164,Z 624.119,A -85,B 0,C 180,E1 -29384.763,E2 -29384.763} C_VEL
LIN {X 0,Y 51.603,Z 625.024,A -85,B 0,C 180,E1 -29387.871,E2 -29387.871} C_VEL
LIN {X 0,Y 45.053,Z 627.598,A -85,B 0,C 180,E1 -29402.082,E2 -29402.082} C_VEL
LIN {X 0,Y 41.502,Z 628.94,A -85,B 0,C 180,E1 -29420.236,E2 -29420.236} C_VEL
LIN {X 0,Y 41.285,Z 629.113,A -85,B 0,C 180,E1 -29429.985,E2 -29429.985} C_VEL
LIN {X 0,Y 42.812,Z 628.479,A -85,B 0,C 180,E1 -29449.151,E2 -29449.151} C_VEL
LIN {X 0,Y 48.079,Z 626.51,A -85,B 0,C 180,E1 -29465.766,E2 -29465.766} C_VEL
LIN {X 0,Y 56.389,Z 623.155,A -85,B 0,C 180,E1 -29478.384,E2 -29478.384} C_VEL
LIN {X 0,Y 66.579,Z 618.312,A -85,B 0,C 180,E1 -29487.597,E2 -29487.597} C_VEL
LIN {X 0,Y 77.952,Z 611.837,A -85,B 0,C 180,E1 -29494.348,E2 -29494.348} C_VEL
LIN {X 0,Y 88.614,Z 604.625,A -85,B 0,C 180,E1 -29498.711,E2 -29498.711} C_VEL
LIN {X 0,Y 99.669,Z 595.695,A -85,B 0,C 180,E1 -29502.14,E2 -29502.14} C_VEL
LIN {X 0,Y 109.396,Z 586.313,A -85,B 0,C 180,E1 -29504.482,E2 -29504.482} C_VEL
LIN {X 0,Y 118.876,Z 575.283,A -85,B 0,C 180,E1 -29506.515,E2 -29506.515} C_VEL
LIN {X 0,Y 127.485,Z 563.17,A -85,B 0,C 180,E1 -29508.078,E2 -29508.078} C_VEL
LIN {X 0,Y 134.194,Z 551.743,A -85,B 0,C 180,E1 -29509.077,E2 -29509.077} C_VEL
LIN {X 0,Y 140.093,Z 539.345,A -85,B 0,C 180,E1 -29509.878,E2 -29509.878} C_VEL
LIN {X 0,Y 144.895,Z 526.37,A -85,B 0,C 180,E1 -29510.521,E2 -29510.521} C_VEL
LIN {X 0,Y 148.718,Z 512.246,A -85,B 0,C 180,E1 -29510.992,E2 -29510.992} C_VEL
LIN {X 0,Y 150.933,Z 499.56,A -85,B 0,C 180,E1 -29511.328,E2 -29511.328} C_VEL
LIN {X 0,Y 150.202,Z 496.444,A -85,B 0,C 180,E1 -29515.076,E2 -29515.076} C_VEL
LIN {X 0,Y 149.921,Z 494.3,A -85,B 0,C 180,E1 -29520,E2 -29520} C_VEL
LIN {X 0,Y 150.286,Z 496.778,A -85,B 0,C 180,E1 -29525.366,E2 -29525.366} C_VEL
LIN {X 0,Y 150.948,Z 499.61,A -85,B 0,C 180,E1 -29528.615,E2 -29528.615} C_VEL
LIN {X 0,Y 148.388,Z 513.924,A -85,B 0,C 180,E1 -29528.984,E2 -29528.984} C_VEL
LIN {X 0,Y 144.447,Z 528.018,A -85,B 0,C 180,E1 -29529.435,E2 -29529.435} C_VEL
LIN {X 0,Y 139.183,Z 541.754,A -85,B 0,C 180,E1 -29530.082,E2 -29530.082} C_VEL
LIN {X 0,Y 133.28,Z 553.768,A -85,B 0,C 180,E1 -29530.88,E2 -29530.88} C_VEL
LIN {X 0,Y 125.715,Z 566.218,A -85,B 0,C 180,E1 -29531.977,E2 -29531.977} C_VEL
LIN {X 0,Y 117.396,Z 577.476,A -85,B 0,C 180,E1 -29533.416,E2 -29533.416} C_VEL
LIN {X 0,Y 109.214,Z 586.838,A -85,B 0,C 180,E1 -29535.171,E2 -29535.171} C_VEL
LIN {X 0,Y 99.478,Z 596.249,A -85,B 0,C 180,E1 -29537.515,E2 -29537.515} C_VEL
LIN {X 0,Y 88.368,Z 605.212,A -85,B 0,C 180,E1 -29540.876,E2 -29540.876} C_VEL
LIN {X 0,Y 77.673,Z 612.457,A -85,B 0,C 180,E1 -29545.221,E2 -29545.221} C_VEL
LIN {X 0,Y 66.247,Z 618.971,A -85,B 0,C 180,E1 -29551.947,E2 -29551.947} C_VEL
LIN {X 0,Y 56.052,Z 623.851,A -85,B 0,C 180,E1 -29561.227,E2 -29561.227} C_VEL
LIN {X 0,Y 47.731,Z 627.239,A -85,B 0,C 180,E1 -29573.932,E2 -29573.932} C_VEL
LIN {X 0,Y 42.579,Z 629.24,A -85,B 0,C 180,E1 -29590.74,E2 -29590.74} C_VEL
LIN {X 0,Y 41.198,Z 629.894,A -85,B 0,C 180,E1 -29610.015,E2 -29610.015} C_VEL
LIN {X 0,Y 42.587,Z 629.202,A -85,B 0,C 180,E1 -29629.287,E2 -29629.287} C_VEL
LIN {X 0,Y 47.743,Z 627.168,A -85,B 0,C 180,E1 -29646.089,E2 -29646.089} C_VEL
LIN {X 0,Y 56.069,Z 623.748,A -85,B 0,C 180,E1 -29658.786,E2 -29658.786} C_VEL
LIN {X 0,Y 61.017,Z 621.489,A -85,B 0,C 180,E1 -29663.748,E2 -29663.748} C_VEL
LIN {X 0,Y 61.946,Z 620.841,A -85,B 0,C 180,E1 -29665.441,E2 -29665.441} C_VEL
LIN {X 0,Y 57.634,Z 618.176,A -85,B 0,C 180,E1 -29692.996,E2 -29692.996} C_VEL
LIN {X 0,Y 75.339,Z 612.948,A -85,B 0,C 180,E1 -29725.912,E2 -29725.912} C_VEL
LIN {X 0,Y 74.715,Z 613.671,A -85,B 0,C 180,E1 -29727.4,E2 -29727.4} C_VEL
LIN {X 0,Y 63.971,Z 619.553,A -85,B 0,C 180,E1 -29734.501,E2 -29734.501} C_VEL
LIN {X 0,Y 56.435,Z 623.034,A -85,B 0,C 180,E1 -29741.636,E2 -29741.636} C_VEL
LIN {X 0,Y 51.603,Z 625.024,A -85,B 0,C 180,E1 -29747.871,E2 -29747.871} C_VEL
LIN {X 0,Y 47.902,Z 626.301,A -85,B 0,C 180,E1 -29753.011,E2 -29753.011} C_VEL
LIN {X 0,Y 41.125,Z 627.888,A -85,B 0,C 180,E1 -29762.162,E2 -29762.162} C_VEL
LIN {X 0,Y 36.445,Z 628.703,A -85,B 0,C 180,E1 -29771.665,E2 -29771.665} C_VEL
LIN {X 0,Y 34.409,Z 629.058,A -85,B 0,C 180,E1 -29780.7,E2 -29780.7} C_VEL
LIN {X 0,Y 34.174,Z 629.092,A -85,B 0,C 180,E1 -29783.988,E2 -29783.988} C_VEL
LIN {X 0,Y 34.175,Z 629.18,A -85,B 0,C 180,E1 -29789.982,E2 -29789.982} C_VEL
LIN {X 0,Y 36.18,Z 628.546,A -85,B 0,C 180,E1 -29812.843,E2 -29812.843} C_VEL
LIN {X 0,Y 42.488,Z 626.578,A -85,B 0,C 180,E1 -29831.406,E2 -29831.406} C_VEL
LIN {X 0,Y 51.932,Z 623.221,A -85,B 0,C 180,E1 -29844.27,E2 -29844.27} C_VEL
LIN {X 0,Y 63.037,Z 618.379,A -85,B 0,C 180,E1 -29853.094,E2 -29853.094} C_VEL
LIN {X 0,Y 75.146,Z 611.903,A -85,B 0,C 180,E1 -29859.243,E2 -29859.243} C_VEL
LIN {X 0,Y 86.286,Z 604.69,A -85,B 0,C 180,E1 -29863.119,E2 -29863.119} C_VEL
LIN {X 0,Y 96.072,Z 597.127,A -85,B 0,C 180,E1 -29865.734,E2 -29865.734} C_VEL
LIN {X 0,Y 106.045,Z 588.046,A -85,B 0,C 180,E1 -29867.803,E2 -29867.803} C_VEL
LIN {X 0,Y 114.388,Z 578.998,A -85,B 0,C 180,E1 -29869.4,E2 -29869.4} C_VEL
LIN {X 0,Y 122.826,Z 568.199,A -85,B 0,C 180,E1 -29870.728,E2 -29870.728} C_VEL
LIN {X 0,Y 130.474,Z 556.38,A -85,B 0,C 180,E1 -29871.762,E2 -29871.762} C_VEL
LIN {X 0,Y 137.309,Z 543.316,A -85,B 0,C 180,E1 -29872.566,E2 -29872.566} C_VEL
LIN {X 0,Y 142.74,Z 529.929,A -85,B 0,C 180,E1 -29873.185,E2 -29873.185} C_VEL
LIN {X 0,Y 146.935,Z 515.882,A -85,B 0,C 180,E1 -29873.613,E2 -29873.613} C_VEL
LIN {X 0,Y 149.282,Z 504.588,A -85,B 0,C 180,E1 -29873.948,E2 -29873.948} C_VEL
LIN {X 0,Y 149.063,Z 503.202,A -85,B 0,C 180,E1 -29875.935,E2 -29875.935} C_VEL
LIN {X 0,Y 148.953,Z 501.46,A -85,B 0,C 180,E1 -29880,E2 -29880} C_VEL
LIN {X 0,Y 149.175,Z 503.756,A -85,B 0,C 180,E1 -29884.898,E2 -29884.898} C_VEL
LIN {X 0,Y 149.302,Z 504.613,A -85,B 0,C 180,E1 -29885.98,E2 -29885.98} C_VEL
LIN {X 0,Y 146.286,Z 518.593,A -85,B 0,C 180,E1 -29886.369,E2 -29886.369} C_VEL
LIN {X 0,Y 142.13,Z 531.767,A -85,B 0,C 180,E1 -29886.751,E2 -29886.751} C_VEL
LIN {X 0,Y 136.397,Z 545.389,A -85,B 0,C 180,E1 -29887.347,E2 -29887.347} C_VEL
LIN {X 0,Y 129.55,Z 558.133,A -85,B 0,C 180,E1 -29888.127,E2 -29888.127} C_VEL
LIN {X 0,Y 121.882,Z 569.722,A -85,B 0,C 180,E1 -29889.117,E2 -29889.117} C_VEL
LIN {X 0,Y 113.185,Z 580.637,A -85,B 0,C 180,E1 -29890.474,E2 -29890.474} C_VEL
LIN {X 0,Y 104.216,Z 590.077,A -85,B 0,C 180,E1 -29892.118,E2 -29892.118} C_VEL
LIN {X 0,Y 94.262,Z 598.911,A -85,B 0,C 180,E1 -29894.272,E2 -29894.272} C_VEL
LIN {X 0,Y 84.471,Z 606.264,A -85,B 0,C 180,E1 -29896.929,E2 -29896.929} C_VEL
LIN {X 0,Y 74.915,Z 612.391,A -85,B 0,C 180,E1 -29900.285,E2 -29900.285} C_VEL
LIN {X 0,Y 62.76,Z 618.904,A -85,B 0,C 180,E1 -29906.404,E2 -29906.404} C_VEL
LIN {X 0,Y 51.618,Z 623.784,A -85,B 0,C 180,E1 -29915.243,E2 -29915.243} C_VEL
LIN {X 0,Y 42.167,Z 627.172,A -85,B 0,C 180,E1 -29928.209,E2 -29928.209} C_VEL
LIN {X 0,Y 35.939,Z 629.172,A -85,B 0,C 180,E1 -29946.995,E2 -29946.995} C_VEL
LIN {X 0,Y 34.092,Z 629.827,A -85,B 0,C 180,E1 -29970.018,E2 -29970.018} C_VEL
LIN {X 0,Y 35.948,Z 629.135,A -85,B 0,C 180,E1 -29993.035,E2 -29993.035} C_VEL
LIN {X 0,Y 42.181,Z 627.099,A -85,B 0,C 180,E1 -30011.813,E2 -30011.813} C_VEL
LIN {X 0,Y 51.637,Z 623.679,A -85,B 0,C 180,E1 -30024.768,E2 -30024.768} C_VEL
LIN {X 0,Y 53.592,Z 622.62,A -85,B 0,C 180,E1 -30028.362,E2 -30028.362} C_VEL
LIN {X 0,Y 50.84,Z 620.805,A -85,B 0,C 180,E1 -30052.055,E2 -30052.055} C_VEL
LIN {X 0,Y 66.039,Z 616.786,A -85,B 0,C 180,E1 -30085.195,E2 -30085.195} C_VEL
LIN {X 0,Y 57.377,Z 620.858,A -85,B 0,C 180,E1 -30090.953,E2 -30090.953} C_VEL
LIN {X 0,Y 46.925,Z 624.977,A -85,B 0,C 180,E1 -30101.49,E2 -30101.49} C_VEL
LIN {X 0,Y 38.899,Z 627.666,A -85,B 0,C 180,E1 -30117.161,E2 -30117.161} C_VEL
LIN {X 0,Y 34.528,Z 629.007,A -85,B 0,C 180,E1 -30138.238,E2 -30138.238} C_VEL
LIN {X 0,Y 34.174,Z 629.092,A -85,B 0,C 180,E1 -30143.988,E2 -30143.988} C_VEL
LIN {X 0,Y 33.789,Z 629.184,A -85,B 0,C 180,E1 -30150.569,E2 -30150.569} C_VEL
LIN {X 0,Y 33.2,Z 629.108,A -85,B 0,C 180,E1 -30157.224,E2 -30157.224} C_VEL
LIN {X 0,Y 32.248,Z 628.757,A -85,B 0,C 180,E1 -30171.065,E2 -30171.065} C_VEL
LIN {X 0,Y 32.922,Z 628.048,A -85,B 0,C 180,E1 -30185.181,E2 -30185.181} C_VEL
LIN {X 0,Y 35.267,Z 627.227,A -85,B 0,C 180,E1 -30194.386,E2 -30194.386} C_VEL
LIN {X 0,Y 36.448,Z 626.888,A -85,B 0,C 180,E1 -30196.919,E2 -30196.919} C_VEL
LIN {X 0,Y 42.513,Z 625.145,A -85,B 0,C 180,E1 -30205.721,E2 -30205.721} C_VEL
LIN {X 0,Y 54,Z 621.061,A -85,B 0,C 180,E1 -30215.619,E2 -30215.619} C_VEL
LIN {X 0,Y 66.456,Z 615.423,A -85,B 0,C 180,E1 -30222.105,E2 -30222.105} C_VEL
LIN {X 0,Y 77.862,Z 609.059,A -85,B 0,C 180,E1 -30225.971,E2 -30225.971} C_VEL
LIN {X 0,Y 89.518,Z 601.145,A -85,B 0,C 180,E1 -30228.883,E2 -30228.883} C_VEL
LIN {X 0,Y 99.664,Z 592.862,A -85,B 0,C 180,E1 -30230.793,E2 -30230.793} C_VEL
LIN {X 0,Y 108.855,Z 583.964,A -85,B 0,C 180,E1 -30232.231,E2 -30232.231} C_VEL
LIN {X 0,Y 117.584,Z 573.916,A -85,B 0,C 180,E1 -30233.503,E2 -30233.503} C_VEL
LIN {X 0,Y 126.187,Z 562.007,A -85,B 0,C 180,E1 -30234.534,E2 -30234.534} C_VEL
LIN {X 0,Y 133.11,Z 550.287,A -85,B 0,C 180,E1 -30235.189,E2 -30235.189} C_VEL
LIN {X 0,Y 139.175,Z 537.479,A -85,B 0,C 180,E1 -30235.744,E2 -30235.744} C_VEL
LIN {X 0,Y 144.082,Z 523.964,A -85,B 0,C 180,E1 -30236.194,E2 -30236.194} C_VEL
LIN {X 0,Y 147.687,Z 510.009,A -85,B 0,C 180,E1 -30236.519,E2 -30236.519} C_VEL
LIN {X 0,Y 147.715,Z 508.52,A -85,B 0,C 180,E1 -30240,E2 -30240} C_VEL
LIN {X 0,Y 147.706,Z 509.951,A -85,B 0,C 180,E1 -30243.367,E2 -30243.367} C_VEL
LIN {X 0,Y 144.146,Z 523.87,A -85,B 0,C 180,E1 -30243.716,E2 -30243.716} C_VEL
LIN {X 0,Y 139.146,Z 537.653,A -85,B 0,C 180,E1 -30244.098,E2 -30244.098} C_VEL
LIN {X 0,Y 133.071,Z 550.478,A -85,B 0,C 180,E1 -30244.605,E2 -30244.605} C_VEL
LIN {X 0,Y 126.148,Z 562.217,A -85,B 0,C 180,E1 -30245.276,E2 -30245.276} C_VEL
LIN {X 0,Y 117.509,Z 574.15,A -85,B 0,C 180,E1 -30246.167,E2 -30246.167} C_VEL
LIN {X 0,Y 108.125,Z 584.882,A -85,B 0,C 180,E1 -30247.469,E2 -30247.469} C_VEL
LIN {X 0,Y 97.855,Z 594.635,A -85,B 0,C 180,E1 -30249.1,E2 -30249.1} C_VEL
LIN {X 0,Y 87.696,Z 602.689,A -85,B 0,C 180,E1 -30251.012,E2 -30251.012} C_VEL
LIN {X 0,Y 76.035,Z 610.411,A -85,B 0,C 180,E1 -30253.98,E2 -30253.98} C_VEL
LIN {X 0,Y 66.257,Z 615.796,A -85,B 0,C 180,E1 -30257.355,E2 -30257.355} C_VEL
LIN {X 0,Y 53.773,Z 621.472,A -85,B 0,C 180,E1 -30263.842,E2 -30263.842} C_VEL
LIN {X 0,Y 42.27,Z 625.59,A -85,B 0,C 180,E1 -30273.792,E2 -30273.792} C_VEL
LIN {X 0,Y 32.824,Z 628.275,A -85,B 0,C 180,E1 -30290.058,E2 -30290.058} C_VEL
LIN {X 0,Y 27.483,Z 629.599,A -85,B 0,C 180,E1 -30315.206,E2 -30315.206} C_VEL
LIN {X 0,Y 27,Z 629.76,A -85,B 0,C 180,E1 -30330.022,E2 -30330.022} C_VEL
LIN {X 0,Y 29.512,Z 629.067,A -85,B 0,C 180,E1 -30358.466,E2 -30358.466} C_VEL
LIN {X 0,Y 37.163,Z 627.031,A -85,B 0,C 180,E1 -30379.176,E2 -30379.176} C_VEL
LIN {X 0,Y 45.224,Z 624.543,A -85,B 0,C 180,E1 -30389.335,E2 -30389.335} C_VEL
LIN {X 0,Y 45.349,Z 624.201,A -85,B 0,C 180,E1 -30392.295,E2 -30392.295} C_VEL
LIN {X 0,Y 45.222,Z 622.472,A -85,B 0,C 180,E1 -30420.001,E2 -30420.001} C_VEL
LIN {X 0,Y 55.151,Z 620.32,A -85,B 0,C 180,E1 -30442.477,E2 -30442.477} C_VEL
LIN {X 0,Y 54.057,Z 620.927,A -85,B 0,C 180,E1 -30444.459,E2 -30444.459} C_VEL
LIN {X 0,Y 42.545,Z 625.045,A -85,B 0,C 180,E1 -30454.292,E2 -30454.292} C_VEL
LIN {X 0,Y 33.125,Z 627.735,A -85,B 0,C 180,E1 -30470.446,E2 -30470.446} C_VEL
LIN {X 0,Y 27.626,Z 629.074,A -85,B 0,C 180,E1 -30495.24,E2 -30495.24} C_VEL
LIN {X 0,Y 27.07,Z 629.247,A -85,B 0,C 180,E1 -30509.978,E2 -30509.978} C_VEL
LIN {X 0,Y 29.742,Z 628.613,A -85,B 0,C 180,E1 -30538.179,E2 -30538.179} C_VEL
LIN {X 0,Y 36.448,Z 626.888,A -85,B 0,C 180,E1 -30556.919,E2 -30556.919} C_VEL
LIN {X 0,Y 39.993,Z 625.839,A -85,B 0,C 180,E1 -30563.843,E2 -30563.843} C_VEL
LIN {X 0,Y 45.652,Z 623.679,A -85,B 0,C 180,E1 -30574.385,E2 -30574.385} C_VEL
LIN {X 0,Y 50.844,Z 621.515,A -85,B 0,C 180,E1 -30581.093,E2 -30581.093} C_VEL
LIN {X 0,Y 55.419,Z 619.626,A -85,B 0,C 180,E1 -30584.606,E2 -30584.606} C_VEL
LIN {X 0,Y 57.082,Z 618.891,A -85,B 0,C 180,E1 -30585.429,E2 -30585.429} C_VEL
LIN {X 0,Y 67.977,Z 613.839,A -85,B 0,C 180,E1 -30589.12,E2 -30589.12} C_VEL
LIN {X 0,Y 79.855,Z 607.049,A -85,B 0,C 180,E1 -30591.874,E2 -30591.874} C_VEL
LIN {X 0,Y 91.861,Z 598.61,A -85,B 0,C 180,E1 -30593.969,E2 -30593.969} C_VEL
LIN {X 0,Y 102.241,Z 589.8,A -85,B 0,C 180,E1 -30595.277,E2 -30595.277} C_VEL
LIN {X 0,Y 112.642,Z 579.127,A -85,B 0,C 180,E1 -30596.534,E2 -30596.534} C_VEL
LIN {X 0,Y 121.349,Z 568.326,A -85,B 0,C 180,E1 -30597.367,E2 -30597.367} C_VEL
LIN {X 0,Y 129.206,Z 556.506,A -85,B 0,C 180,E1 -30597.998,E2 -30597.998} C_VEL
LIN {X 0,Y 136.202,Z 543.439,A -85,B 0,C 180,E1 -30598.501,E2 -30598.501} C_VEL
LIN {X 0,Y 141.478,Z 530.814,A -85,B 0,C 180,E1 -30598.875,E2 -30598.875} C_VEL
LIN {X 0,Y 145.811,Z 516.945,A -85,B 0,C 180,E1 -30599.138,E2 -30599.138} C_VEL
LIN {X 0,Y 146.08,Z 515.813,A -85,B 0,C 180,E1 -30599.225,E2 -30599.225} C_VEL
LIN {X 0,Y 146.133,Z 515.553,A -85,B 0,C 180,E1 -30600,E2 -30600} C_VEL
LIN {X 0,Y 146.077,Z 515.846,A -85,B 0,C 180,E1 -30600.694,E2 -30600.694} C_VEL
LIN {X 0,Y 142.13,Z 528.975,A -85,B 0,C 180,E1 -30600.973,E2 -30600.973} C_VEL
LIN {X 0,Y 137.068,Z 541.571,A -85,B 0,C 180,E1 -30601.285,E2 -30601.285} C_VEL
LIN {X 0,Y 130.941,Z 553.581,A -85,B 0,C 180,E1 -30601.684,E2 -30601.684} C_VEL
LIN {X 0,Y 123.071,Z 566.029,A -85,B 0,C 180,E1 -30602.233,E2 -30602.233} C_VEL
LIN {X 0,Y 114.344,Z 577.283,A -85,B 0,C 180,E1 -30602.942,E2 -30602.942} C_VEL
LIN {X 0,Y 105.654,Z 586.644,A -85,B 0,C 180,E1 -30603.91,E2 -30603.91} C_VEL
LIN {X 0,Y 95.255,Z 596.054,A -85,B 0,C 180,E1 -30605.18,E2 -30605.18} C_VEL
LIN {X 0,Y 83.18,Z 605.014,A -85,B 0,C 180,E1 -30606.956,E2 -30606.956} C_VEL
LIN {X 0,Y 71.234,Z 612.259,A -85,B 0,C 180,E1 -30609.446,E2 -30609.446} C_VEL
LIN {X 0,Y 57.838,Z 618.771,A -85,B 0,C 180,E1 -30613.616,E2 -30613.616} C_VEL
LIN {X 0,Y 44.915,Z 623.65,A -85,B 0,C 180,E1 -30620.182,E2 -30620.182} C_VEL
LIN {X 0,Y 32.925,Z 627.038,A -85,B 0,C 180,E1 -30631.408,E2 -30631.408} C_VEL
LIN {X 0,Y 23.48,Z 629.038,A -85,B 0,C 180,E1 -30653.26,E2 -30653.26} C_VEL
LIN {X 0,Y 19.897,Z 629.692,A -85,B 0,C 180,E1 -30690.03,E2 -30690.03} C_VEL
LIN {X 0,Y 23.493,Z 628.999,A -85,B 0,C 180,E1 -30726.78,E2 -30726.78} C_VEL
LIN {X 0,Y 32.943,Z 626.963,A -85,B 0,C 180,E1 -30748.612,E2 -30748.612} C_VEL
LIN {X 0,Y 36.994,Z 625.941,A -85,B 0,C 180,E1 -30753.285,E2 -30753.285} C_VEL
LIN {X 0,Y 37.426,Z 625.527,A -85,B 0,C 180,E1 -30757.941,E2 -30757.941} C_VEL
LIN {X 0,Y 40.698,Z 623.949,A -85,B 0,C 180,E1 -30789.945,E2 -30789.945} C_VEL
LIN {X 0,Y 44.653,Z 623.253,A -85,B 0,C 180,E1 -30799.167,E2 -30799.167} C_VEL
LIN {X 0,Y 45.159,Z 623.239,A -85,B 0,C 180,E1 -30800.933,E2 -30800.933} C_VEL
LIN {X 0,Y 33.178,Z 626.631,A -85,B 0,C 180,E1 -30812.047,E2 -30812.047} C_VEL
LIN {X 0,Y 23.725,Z 628.638,A -85,B 0,C 180,E1 -30833.638,E2 -30833.638} C_VEL
LIN {X 0,Y 19.98,Z 629.315,A -85,B 0,C 180,E1 -30869.97,E2 -30869.97} C_VEL
LIN {X 0,Y 23.708,Z 628.68,A -85,B 0,C 180,E1 -30906.329,E2 -30906.329} C_VEL
LIN {X 0,Y 33.151,Z 626.712,A -85,B 0,C 180,E1 -30927.96,E2 -30927.96} C_VEL
LIN {X 0,Y 45.121,Z 623.355,A -85,B 0,C 180,E1 -30939.115,E2 -30939.115} C_VEL
LIN {X 0,Y 57.082,Z 618.891,A -85,B 0,C 180,E1 -30945.429,E2 -30945.429} C_VEL
LIN {X 0,Y 61.917,Z 616.724,A -85,B 0,C 180,E1 -30947.966,E2 -30947.966} C_VEL
LIN {X 0,Y 69.357,Z 612.844,A -85,B 0,C 180,E1 -30952.634,E2 -30952.634} C_VEL
LIN {X 0,Y 76.935,Z 608.482,A -85,B 0,C 180,E1 -30956.245,E2 -30956.245} C_VEL
LIN {X 0,Y 81.779,Z 605.444,A -85,B 0,C 180,E1 -30957.312,E2 -30957.312} C_VEL
LIN {X 0,Y 93.139,Z 597.323,A -85,B 0,C 180,E1 -30958.545,E2 -30958.545} C_VEL
LIN {X 0,Y 104.072,Z 587.856,A -85,B 0,C 180,E1 -30959.452,E2 -30959.452} C_VEL
LIN {X 0,Y 105.411,Z 586.571,A -85,B 0,C 180,E1 -30959.55,E2 -30959.55} C_VEL
LIN {X 0,Y 105.763,Z 586.219,A -85,B 0,C 180,E1 -30960,E2 -30960} C_VEL
LIN {X 0,Y 94.878,Z 595.989,A -85,B 0,C 180,E1 -30960.894,E2 -30960.894} C_VEL
LIN {X 0,Y 82.62,Z 604.949,A -85,B 0,C 180,E1 -30962.048,E2 -30962.048} C_VEL
LIN {X 0,Y 70.417,Z 612.193,A -85,B 0,C 180,E1 -30963.72,E2 -30963.72} C_VEL
LIN {X 0,Y 60.023,Z 617.271,A -85,B 0,C 180,E1 -30965.7,E2 -30965.7} C_VEL
LIN {X 0,Y 46.355,Z 622.515,A -85,B 0,C 180,E1 -30969.859,E2 -30969.859} C_VEL
LIN {X 0,Y 36.325,Z 625.456,A -85,B 0,C 180,E1 -30974.744,E2 -30974.744} C_VEL
LIN {X 0,Y 23.715,Z 628.141,A -85,B 0,C 180,E1 -30987.304,E2 -30987.304} C_VEL
LIN {X 0,Y 14.195,Z 629.465,A -85,B 0,C 180,E1 -31020.373,E2 -31020.373} C_VEL
LIN {X 0,Y 12.786,Z 629.625,A -85,B 0,C 180,E1 -31050.047,E2 -31050.047} C_VEL
LIN {X 0,Y 18.295,Z 628.931,A -85,B 0,C 180,E1 -31100.253,E2 -31100.253} C_VEL
LIN {X 0,Y 29.857,Z 626.895,A -85,B 0,C 180,E1 -31120.372,E2 -31120.372} C_VEL
LIN {X 0,Y 30.027,Z 626.645,A -85,B 0,C 180,E1 -31126.465,E2 -31126.465} C_VEL
LIN {X 0,Y 34.476,Z 625.629,A -85,B 0,C 180,E1 -31154.501,E2 -31154.501} C_VEL
LIN {X 0,Y 32.196,Z 626.205,A -85,B 0,C 180,E1 -31158.54,E2 -31158.54} C_VEL
LIN {X 0,Y 23.92,Z 627.871,A -85,B 0,C 180,E1 -31168.131,E2 -31168.131} C_VEL
LIN {X 0,Y 14.354,Z 629.209,A -85,B 0,C 180,E1 -31200.636,E2 -31200.636} C_VEL
LIN {X 0,Y 12.878,Z 629.382,A -85,B 0,C 180,E1 -31229.953,E2 -31229.953} C_VEL
LIN {X 0,Y 18.468,Z 628.747,A -85,B 0,C 180,E1 -31279.51,E2 -31279.51} C_VEL
LIN {X 0,Y 29.981,Z 626.779,A -85,B 0,C 180,E1 -31299.601,E2 -31299.601} C_VEL
LIN {X 0,Y 43.095,Z 623.422,A -85,B 0,C 180,E1 -31308.024,E2 -31308.024} C_VEL
LIN {X 0,Y 56.826,Z 618.507,A -85,B 0,C 180,E1 -31312.895,E2 -31312.895} C_VEL
LIN {X 0,Y 70.465,Z 612.101,A -85,B 0,C 180,E1 -31315.716,E2 -31315.716} C_VEL
LIN {X 0,Y 81.779,Z 605.444,A -85,B 0,C 180,E1 -31317.312,E2 -31317.312} C_VEL
LIN {X 0,Y 80.201,Z 606.442,A -85,B 0,C 180,E1 -31317.869,E2 -31317.869} C_VEL
LIN {X 0,Y 71.415,Z 611.555,A -85,B 0,C 180,E1 -31318.572,E2 -31318.572} C_VEL
LIN {X 0,Y 60.267,Z 616.971,A -85,B 0,C 180,E1 -31318.776,E2 -31318.776} C_VEL
LIN {X 0,Y 48.794,Z 621.431,A -85,B 0,C 180,E1 -31318.443,E2 -31318.443} C_VEL
LIN {X 0,Y 40.985,Z 623.81,A -85,B 0,C 180,E1 -31317.309,E2 -31317.309} C_VEL
LIN {X 0,Y 28.296,Z 626.846,A -85,B 0,C 180,E1 -31313.269,E2 -31313.269} C_VEL
LIN {X 0,Y 14.862,Z 628.815,A -85,B 0,C 180,E1 -31300.915,E2 -31300.915} C_VEL
LIN {X 0,Y 5.77,Z 629.449,A -85,B 0,C 180,E1 -31229.895,E2 -31229.895} C_VEL
LIN {X 0,Y 14.884,Z 628.774,A -85,B 0,C 180,E1 -31159.077,E2 -31159.077} C_VEL
LIN {X 0,Y 21.5,Z 627.939,A -85,B 0,C 180,E1 -31151.151,E2 -31151.151} C_VEL
LIN {X 0,Y 24.431,Z 627.439,A -85,B 0,C 180,E1 -31144.882,E2 -31144.882} C_VEL
LIN {X 0,Y 23.782,Z 627.548,A -85,B 0,C 180,E1 -31140.001,E2 -31140.001} C_VEL
LIN {X 0,Y 21.421,Z 628.014,A -85,B 0,C 180,E1 -31129.978,E2 -31129.978} C_VEL
LIN {X 0,Y 8.774,Z 629.378,A -85,B 0,C 180,E1 -31103.34,E2 -31103.34} C_VEL
LIN {X 0,Y 5.688,Z 629.558,A -85,B 0,C 180,E1 -31050.106,E2 -31050.106} C_VEL
LIN {X 0,Y 8.757,Z 629.397,A -85,B 0,C 180,E1 -30996.741,E2 -30996.741} C_VEL
LIN {X 0,Y 21.4,Z 628.073,A -85,B 0,C 180,E1 -30970.032,E2 -30970.032} C_VEL
LIN {X 0,Y 35.193,Z 625.39,A -85,B 0,C 180,E1 -30963.452,E2 -30963.452} C_VEL
LIN {X 0,Y 49.185,Z 621.271,A -85,B 0,C 180,E1 -30960.291,E2 -30960.291} C_VEL
LIN {X 0,Y 50.82,Z 620.691,A -85,B 0,C 180,E1 -30959.999,E2 -30959.999} C_VEL
LIN {X 0,Y 49.193,Z 621.26,A -85,B 0,C 180,E1 -30958.932,E2 -30958.932} C_VEL
LIN {X 0,Y 40.985,Z 623.81,A -85,B 0,C 180,E1 -30957.309,E2 -30957.309} C_VEL
LIN {X 0,Y 40.985,Z 623.81,A -85,B 0,C 180,E1 -30957.309,E2 -30957.309}

QRS_NEXT_CUT()

QRS_NEXT()
QRS_HOME()

END
